(* IEC 61131-3 sources: elnaProjects/ElpcLogic/PomarKc7Unchanged/build_USO_ecl, 1 file *)

(* ---- plc.st ---- *)
TYPE
  TItemAIN : STRUCT
    wFlags : UINT := 0;
    wReserved : UINT := 0;
    dblValue : LREAL := 0.0;
    nanosec : ULINT := 0;
    reserve : ULINT := 0;
  END_STRUCT;
  TYPE_ReliableBit : STRUCT
    value : BOOL;
    reliability : BOOL;
    _inversed : BOOL;
  END_STRUCT;
  TItemDIN : STRUCT
    wFlags : UINT := 0;
    wValue : UINT := 0;
    nanosec : ULINT := 0;
    reserve : ULINT := 0;
  END_STRUCT;
  struct_DI : STRUCT
    imit : BOOL;
    value : WORD;
    reliability : WORD;
    bits : ARRAY [0..15] OF TYPE_ReliableBit;
    blConnect : BOOL;
  END_STRUCT;
  TYPE_StatusAi : STRUCT
    NOTDEFINED : BYTE := 0;
    LL : BYTE := 1;
    HL : BYTE := 2;
    NOTRELIABLE : BYTE := 3;
    normal : BYTE := 4;
    LW : BYTE := 5;
    HW : BYTE := 6;
    LA : BYTE := 7;
    HA : BYTE := 8;
  END_STRUCT;
  TWordData : STRUCT
    wFlags : UINT := 0;
    wValue : UINT := 0;
  END_STRUCT;
  TDoubleData : STRUCT
    wFlags : UINT := 0;
    dblValue : LREAL := 0.0;
  END_STRUCT;
  TYPE_statusDualInput : STRUCT
    STATUS_NOTDEFINED : BYTE := 0;
    STATUS_ON : BYTE := 1;
    STATUS_OFF : BYTE := 2;
    STATUS_TRANSITIONAL : BYTE := 3;
    STATUS_ERROR : BYTE := 4;
  END_STRUCT;
  TYPE_CommandAnalog : STRUCT
    cmd_SetUstavki : WORD := 1;
    cmd_SetRemont : WORD := 2;
    cmd_ResetRemont : WORD := 3;
    cmd_kvitNotReliable : WORD := 4;
  END_STRUCT;
  struct_AI : STRUCT
    value : LREAL;
    status : DWORD;
    interval : BYTE;
    inCommand : WORD;
    blConnect : BOOL;
    dLL : LREAL;
    dHL : LREAL;
    dLA : LREAL;
    dHA : LREAL;
    dLW : LREAL;
    dHW : LREAL;
    LL : LREAL;
    HL : LREAL;
    LA : LREAL;
    HA : LREAL;
    LW : LREAL;
    HW : LREAL;
    ISVALIDREF_LA : BOOL;
    ISVALIDREF_HA : BOOL;
    ISVALIDREF_LW : BOOL;
    ISVALIDREF_HW : BOOL;
    inpLL : LREAL;
    inpHL : LREAL;
    CurrentShotCircuit : LREAL;
    CurrentBreakCircuit : LREAL;
    maxChangeSpeed : LREAL;
    maxChangeSpeedDown : LREAL;
    ChangeSpeed : LREAL;
    histeresis : LREAL;
    aperturFilter : LREAL;
    exponentialFilter : LREAL;
    rassoglasovanie : LREAL;
    OpcCommandsDisabled : BOOL;
    Disabled_LA : BOOL;
    Disabled_HA : BOOL;
    Disabled_LW : BOOL;
    Disabled_HW : BOOL;
    delayLA : TIME;
    delayLW : TIME;
    delayHW : TIME;
    delayHA : TIME;
    minValue_ISVALIDREF : BOOL;
    maxValue_ISVALIDREF : BOOL;
    minValue : LREAL;
    maxValue : LREAL;
    inOpcCommandsDisabled : BOOL;
    imit : BOOL;
    remont : BOOL;
    NS : BOOL;
    NS_Min : BOOL;
    NS_Max : BOOL;
    inCommand_Alg : WORD;
    inCommand_ARM : WORD;
    dMaxChangeSpeed : LREAL;
    dMaxChangeSpeedDown : LREAL;
  END_STRUCT;
  AiConfig : STRUCT
    T_obmotki_fazy_1_k : struct_AI;
    T_aktivnogo_zheleza_statora_1_k : struct_AI;
    T_obmotki_fazy_2_k : struct_AI;
    T_aktivnogo_zheleza_statora_2_k : struct_AI;
    T_obmotki_fazy_3_k : struct_AI;
    T_aktivnogo_zheleza_statora_3_k : struct_AI;
    T_masla_v_maslobake : struct_AI;
    T_perednego_opornogo_podshipnika_dvigatelia_t1 : struct_AI;
    T_zadnego_opornogo_podshipnika_dvigatelia_t2 : struct_AI;
    T_masla_na_slive_perednego_opornogo_podshipnika_dvigatelia : struct_AI;
    T_masla_na_slive_zadnego_opornogo_podshipnika_dvigatelia : struct_AI;
    T_podshipnika_reduktora_t1 : struct_AI;
    T_podshipnika_reduktora_t2 : struct_AI;
    T_podshipnika_reduktora_t3 : struct_AI;
    T_podshipnika_reduktora_t4 : struct_AI;
    T_opornogo_podshipnika_nagnetatelia_t1 : struct_AI;
    T_opornogo_podshipnika_nagnetatelia_t2 : struct_AI;
    T_opornogo_podshipnika_nagnetatelia_t3 : struct_AI;
    T_oporno_upornogo_podshipnika_nagnetatelia_t4 : struct_AI;
    T_masla_do_AVOM : struct_AI;
    T_masla_posle_AVOM : struct_AI;
    T_gaz_in_nagnetatelia : struct_AI;
    T_gaz_out_nagnetatelia : struct_AI;
    T_hotAir_dvigatelia_t1 : struct_AI;
    T_clodAir_dvigatelia_t1 : struct_AI;
    dPmaslo_gaz : struct_AI;
    dP_gaza_na_konfuzore_nagnetatelia : struct_AI;
    P_masla_uplotneniia : struct_AI;
    P_gaza_na_vkhode_nagnetatelia : struct_AI;
    P_gaza_na_vykhode_nagnetatelia : struct_AI;
    P_masla_smazki_nizkoe : struct_AI;
    P_masla_smazki_srednee_posle_nasosov : struct_AI;
    Vibratciia_STD_t1 : struct_AI;
    Vibratciia_STD_t2 : struct_AI;
    Vibratciia_rotora_nagnetatelia_t1 : struct_AI;
    Vibratciia_rotora_nagnetatelia_t2 : struct_AI;
    Vibratciia_rotora_nagnetatelia_t3 : struct_AI;
    Vibratciia_rotora_nagnetatelia_t4 : struct_AI;
    Osevoi_sdvig_rotora_nagnetatelia : struct_AI;
    Uroven_masla_v_maslobake : struct_AI;
    Tok_vozbuzhdeniia_vozbuditelia : struct_AI;
    Tok_statora_elektrodvigatelia : struct_AI;
    Aktivnaia_moshchnost : struct_AI;
    Reaktivnaia_moshchnost : struct_AI;
    VoltageSHU_osnovnoi_vvod : struct_AI;
    VoltageSHU_rezervnyi_vvod : struct_AI;
    Rashod : struct_AI;
    Zapas : struct_AI;
    T_vnytri_shkafa : struct_AI;
  END_STRUCT;
  TYPE_AnalogLimitFlags : STRUCT
    NONE : BYTE := 0;
    LL : BYTE := 16#1;
    LW : BYTE := 16#2;
    HW : BYTE := 16#4;
    LA : BYTE := 16#8;
    HA : BYTE := 16#10;
    HL : BYTE := 16#20;
    SipUP : BYTE := 16#40;
    SipDown : BYTE := 16#80;
  END_STRUCT;
  DiConfig : STRUCT
    di_0 : struct_DI;
    di_1 : struct_DI;
    di_2 : struct_DI;
    di_3 : struct_DI;
    di_4 : struct_DI;
    di_5 : struct_DI;
    di_6 : struct_DI;
    di_7 : struct_DI;
    di_8 : struct_DI;
    di_9 : struct_DI;
    di_10 : struct_DI;
    di_11 : struct_DI;
    di_12 : struct_DI;
    di_13 : struct_DI;
    di_14 : struct_DI;
    di_15 : struct_DI;
  END_STRUCT;
  TYPE_commandDualInput : STRUCT
    CMD_ON : BYTE := 1;
    CMD_OFF : BYTE := 2;
    CMD_RESET : BYTE := 3;
  END_STRUCT;
  struct_DO : STRUCT
    imit : BOOL;
    blConnect : BOOL;
    value : WORD;
    bits : ARRAY [0..15] OF BOOL;
  END_STRUCT;
  DOconfig : STRUCT
    do_0 : struct_DO;
    do_1 : struct_DO;
    do_2 : struct_DO;
    do_3 : struct_DO;
    do_4 : struct_DO;
    do_5 : struct_DO;
    do_6 : struct_DO;
    do_7 : struct_DO;
    gpio_out : struct_DO;
  END_STRUCT;
  struct_AO : STRUCT
    nValue : LREAL;
    blConnect : BOOL;
    outLL : LREAL;
    outHL : LREAL;
    newLL : LREAL;
    newHL : LREAL;
    newLL_ISVALIDREF : BOOL;
    newHL_ISVALIDREF : BOOL;
    inCommand : WORD;
    Value : LREAL;
    status : DWORD;
    LL : LREAL;
    HL : LREAL;
    OpcCommandsDisabled : BOOL;
  END_STRUCT;
  AOConfig : STRUCT
    Reserv_AO_1 : struct_AO;
    Reserv_AO_2 : struct_AO;
  END_STRUCT;
  struct_singleSignal : STRUCT
    reliability : BOOL;
    inverse : BOOL;
    DelayOn : TIME;
    DelayOff : TIME;
    Q : BOOL;
    status : DWORD;
    Disabled_Sig : BOOL;
  END_STRUCT;
  IM_singleSignals : STRUCT
    dP_gazgaz_Kran1 : struct_singleSignal;
    OsevoiSdvig_pravo : struct_singleSignal;
    OsevoiSdvig_levo : struct_singleSignal;
    dP_oilgaz_low : struct_singleSignal;
    P_oil_low : struct_singleSignal;
    KZ_10kv : struct_singleSignal;
    Vozb_ProboiVentila : struct_singleSignal;
    Vozb_AsinchHod : struct_singleSignal;
    Vozb_ReSynchronize : struct_singleSignal;
    Vozb_ControlVozbuditela : struct_singleSignal;
    NS_ForsingVozbugdenia : struct_singleSignal;
    NS_Vozbyditela : struct_singleSignal;
    Vozb_AVR_off : struct_singleSignal;
    Vozb_AutoUprVozbuditela_off : struct_singleSignal;
    Vozb_KontaktorON : struct_singleSignal;
    Vozb_Overload : struct_singleSignal;
    AO_KC : struct_singleSignal;
    AOGPA_PRU : struct_singleSignal;
    BEO_Ready : struct_singleSignal;
    BEO_Srabat : struct_singleSignal;
    BEO_ON_knopkaSHU : struct_singleSignal;
    BEO_ON_knopkaPRU : struct_singleSignal;
    NOGPA_knopkaSHU : struct_singleSignal;
    AOGPA_knopkaSHU : struct_singleSignal;
    DverShkafaOtkryta : struct_singleSignal;
    QF1_on : struct_singleSignal;
    QF2_on : struct_singleSignal;
    QF23_on : struct_singleSignal;
    QF4_QF5_on : struct_singleSignal;
    QF6_QF7_on : struct_singleSignal;
    QF8_QF9_on : struct_singleSignal;
    QF10_QF11_on : struct_singleSignal;
    QF12_QF13_on : struct_singleSignal;
    QF14_QF15_on : struct_singleSignal;
    QF22_on : struct_singleSignal;
    NS_G1_G2 : struct_singleSignal;
    NS_G3_G4 : struct_singleSignal;
    NS_G15_G16 : struct_singleSignal;
    NS_G17 : struct_singleSignal;
    NS_G5_G6 : struct_singleSignal;
    NS_G7_G8 : struct_singleSignal;
    NS_G18_G19 : struct_singleSignal;
    NS_G10_G11 : struct_singleSignal;
    NS_G13_G14 : struct_singleSignal;
  END_STRUCT;
  struct_singleOutput : STRUCT
    wait_time : TIME;
    inCommand : WORD;
    inOpcCommandsDisabled : BOOL;
    Q : BOOL;
    status : DWORD;
    OpcCommandsDisabled : BOOL;
    inCommand_Alg : WORD;
    inCommand_ARM : WORD;
  END_STRUCT;
  IM_singleOutputs : STRUCT
    Lampa_NO : struct_singleOutput;
    VzvodBREO : struct_singleOutput;
    AO_GPA : struct_singleOutput;
    SbrosBREO : struct_singleOutput;
    IndikicijaPS_fonar : struct_singleOutput;
    IndikicijaAS_fonar : struct_singleOutput;
    mv_off_KNA : struct_singleOutput;
  END_STRUCT;
  struct_Kran : STRUCT
    inCommand : WORD;
    status : DWORD;
    onStatus : BYTE;
    inOpcCommandsDisabled : BOOL;
    sdvig : BOOL;
    Ns : BOOL;
    Dp : BOOL;
    CommandFault : BOOL;
    Accident : BOOL;
    Auto : BOOL;
    Manual : BOOL;
    Local : BOOL;
    Distance : BOOL;
    ErrorPowerOff : BOOL;
    ErrorBlock : BOOL;
    So : BOOL;
    Sz : BOOL;
    OpcCommandsDisabled : BOOL;
    lastCmdIsOn : BOOL;
    ISVALIDREF_statOn : BOOL;
    ISVALIDREF_statOff : BOOL;
    ISVALIDREF_cmdOn : BOOL;
    ISVALIDREF_cmdOff : BOOL;
    ISVALIDREF_inSo : BOOL;
    ISVALIDREF_inSz : BOOL;
    ISVALIDREF_inDp : BOOL;
    continueHoldCommand : TIME;
    inCommand_Alg : WORD;
    inCommand_ARM : WORD;
    cmdOn : BOOL;
    cmdOff : BOOL;
    reliability : BOOL;
  END_STRUCT;
  struct_OilPump : STRUCT
    inCommand : WORD;
    inCommand_Alg : WORD;
    inCommand_ARM : WORD;
    status : DWORD;
    onStatus : BYTE;
    inOpcCommandsDisabled : BOOL;
    sdvig : BOOL;
    Ns : BOOL;
    CommandFault : BOOL;
    Accident : BOOL;
    Local : BOOL;
    Distance : BOOL;
    BreakCmdOn : BOOL;
    BreakCmdOff : BOOL;
    OpcCommandsDisabled : BOOL;
    lastCmdIsOn : BOOL;
    ISVALIDREF_statOn : BOOL;
    ISVALIDREF_statOff : BOOL;
    ISVALIDREF_cmdOn : BOOL;
    ISVALIDREF_cmdOff : BOOL;
    ISVALIDREF_inBreakCmdOn : BOOL;
    ISVALIDREF_inBreakCmdOff : BOOL;
    inBlocked : BOOL;
    Blocked : BOOL;
    Osnovnoy : BOOL;
    Rezervny : BOOL;
    cmdOn : BOOL;
    cmdOff : BOOL;
    reliability : BOOL;
  END_STRUCT;
  struct_Switch : STRUCT
    inCommand : WORD;
    status : DWORD;
    onStatus : BYTE;
    inOpcCommandsDisabled : BOOL;
    sdvig : BOOL;
    Ns : BOOL;
    CommandFault : BOOL;
    Accident : BOOL;
    Auto : BOOL;
    Manual : BOOL;
    Local : BOOL;
    Distance : BOOL;
    ErrorPowerOff : BOOL;
    ErrorBlock : BOOL;
    BreakCmdOn : BOOL;
    BreakCmdOff : BOOL;
    OpcCommandsDisabled : BOOL;
    lastCmdIsOn : BOOL;
    ISVALIDREF_statOn : BOOL;
    ISVALIDREF_statOff : BOOL;
    ISVALIDREF_cmdOn : BOOL;
    ISVALIDREF_cmdOff : BOOL;
    ISVALIDREF_inBreakCmdOn : BOOL;
    ISVALIDREF_inBreakCmdOff : BOOL;
    inCommand_Alg : WORD;
    inCommand_ARM : WORD;
    cmdOn : BOOL;
    cmdOff : BOOL;
    reliability : BOOL;
  END_STRUCT;
  struct_SectionSwitch : STRUCT
    inCommand : WORD;
    status : DWORD;
    onStatus : BYTE;
    inOpcCommandsDisabled : BOOL;
    sdvig : BOOL;
    Ns : BOOL;
    CommandFault : BOOL;
    Accident : BOOL;
    Local : BOOL;
    Distance : BOOL;
    OpcCommandsDisabled : BOOL;
    lastCmdIsOn : BOOL;
    offKNA : BOOL;
    basketStatus : BYTE;
    ISVALIDREF_statOn : BOOL;
    ISVALIDREF_statOff : BOOL;
    ISVALIDREF_cmdOn : BOOL;
    ISVALIDREF_cmdOff : BOOL;
    ISVALIDREF_inBreakCmdOn : BOOL;
    ISVALIDREF_inBreakCmdOff : BOOL;
    BreakCmdOn : BOOL;
    BreakCmdOff : BOOL;
    ISVALIDREF_basketRolledIn : BOOL;
    ISVALIDREF_basketRolledOut : BOOL;
    ISVALIDREF_basketTest : BOOL;
    inCommand_Alg : WORD;
    inCommand_ARM : WORD;
    cmdOn : BOOL;
    cmdOff : BOOL;
    reliability : BOOL;
  END_STRUCT;
  struct_ReserveIM : STRUCT
    var1 : BOOL;
    var2 : BOOL;
  END_STRUCT;
  struct_ReserveIM2 : STRUCT
    var1 : BOOL;
    var2 : BOOL;
  END_STRUCT;
  struct_AnalogParametr : STRUCT
    inCommand : WORD;
    inCommand_Alg : WORD;
    inCommand_ARM : WORD;
    status : DWORD;
    newValue : LREAL;
    currentValue : LREAL;
    minVal : LREAL;
    maxVal : LREAL;
    maxStep : LREAL;
    minVal_ISVALIDREF : BOOL;
    maxVal_ISVALIDREF : BOOL;
    maxStep_ISVALIDREF : BOOL;
    inOpcCommandsDisabled : BOOL;
    Value : LREAL;
    isValidValue : BOOL;
    OpcCommandsDisabled : BOOL;
  END_STRUCT;
  struct_DiscretParametr : STRUCT
    newValue : UINT;
    currentValue : UINT;
    inOpcCommandsDisabled : BOOL;
    inCommand : WORD;
    inCommand_Alg : WORD;
    inCommand_ARM : WORD;
    status : DWORD;
    OpcCommandsDisabled : BOOL;
    Value : UINT;
  END_STRUCT;
  ImConfig : STRUCT
    Kran1 : struct_Kran;
    Kran2 : struct_Kran;
    Kran3b : struct_Kran;
    Kran4 : struct_Kran;
    Kran5 : struct_Kran;
    Kran6 : struct_Kran;
    nu1 : struct_OilPump;
    nu2 : struct_OilPump;
    pns : struct_Switch;
    v1_Avom : struct_Switch;
    v2_Avom : struct_Switch;
    mv : struct_SectionSwitch;
    Ten : struct_Switch;
    Reserve_IM1 : struct_ReserveIM;
    Reserve_IM2 : struct_ReserveIM2;
    SingleSignals : IM_singleSignals;
    SingleOutputs : IM_singleOutputs;
    AutoAvom_onTemp1 : struct_AnalogParametr;
    AutoAvom_onTemp2 : struct_AnalogParametr;
    AutoAvom_hysteresis : struct_AnalogParametr;
    TypeSwitch : struct_DiscretParametr;
    AutoPns_UstRun : struct_AnalogParametr;
    AutoPns_UstStop : struct_AnalogParametr;
    AutoNU_mainNU : struct_DiscretParametr;
    PuskOilSystem_UstdPmg : struct_AnalogParametr;
    AutoTen_offTemperature : struct_AnalogParametr;
    AutoNU_Ust_Swap : struct_AnalogParametr;
    testdPmg_Ust_dPLow : struct_AnalogParametr;
    AntiPompag_UgolVNA : struct_AnalogParametr;
    AntiPompag_K : struct_AnalogParametr;
    AntiPompag_A : struct_AnalogParametr;
    AntiPompag_y0 : struct_AnalogParametr;
  END_STRUCT;
  struct_DualStateIm : STRUCT
    inCommand : WORD;
    status : DWORD;
    onStatus : BYTE;
    inOpcCommandsDisabled : BOOL;
    sdvig : BOOL;
    Ns : BOOL;
    CommandFault : BOOL;
    Accident : BOOL;
    OpcCommandsDisabled : BOOL;
    lastCmdIsOn : BOOL;
    ISVALIDREF_statOn : BOOL;
    ISVALIDREF_statOff : BOOL;
    ISVALIDREF_cmdOn : BOOL;
    ISVALIDREF_cmdOff : BOOL;
    inCommand_Alg : WORD;
    inCommand_ARM : WORD;
    cmdOn : BOOL;
    cmdOff : BOOL;
    reliability : BOOL;
  END_STRUCT;
  TYPE_ProtectionTags : STRUCT
    NOTHING : BYTE := 0;
    AOB : BYTE := 1;
    AOS : BYTE := 2;
    AOPOJ : BYTE := 3;
  END_STRUCT;
  TYPE_basketStats : STRUCT
    BASKET_NOTDEFINED : BYTE := 0;
    BASKET_ROLLEDIN : BYTE := 1;
    BASKET_ROLLEDOUT : BYTE := 2;
    BASKET_TRANSITIONAL : BYTE := 3;
    BASKET_ERROR : BYTE := 4;
    BASKET_TEST : BYTE := 5;
  END_STRUCT;
  struct_AiProtection : STRUCT
    controlLimit : BYTE;
    delay : TIME;
    inTag : BYTE;
    inRunOnStart : BOOL;
    inCanRun : BOOL;
    inOpcCommandsDisabled : BOOL;
    inCommand : WORD;
    inCommand_Alg : WORD;
    inCommand_ARM : WORD;
    Tag : BYTE;
    status : DWORD;
    CanRun : BOOL;
    OpcCommandsDisabled : BOOL;
    isRunning : BOOL;
    HasError : BOOL;
    isEnded : BOOL;
    Remont : BOOL;
    Check : BOOL;
    Signaling : BOOL;
    SignalingTP : BOOL;
    RunOnStart : BOOL;
  END_STRUCT;
  struct_DiProtection : STRUCT
    delay : TIME;
    inTag : BYTE;
    inRunOnStart : BOOL;
    inCanRun : BOOL;
    inOpcCommandsDisabled : BOOL;
    inCommand : WORD;
    inCommand_Alg : WORD;
    inCommand_ARM : WORD;
    Tag : BYTE;
    status : DWORD;
    CanRun : BOOL;
    OpcCommandsDisabled : BOOL;
    isRunning : BOOL;
    HasError : BOOL;
    isEnded : BOOL;
    Remont : BOOL;
    Check : BOOL;
    Signaling : BOOL;
    SignalingTP : BOOL;
    RunOnStart : BOOL;
  END_STRUCT;
  ProtectionsConfig : STRUCT
    T_perednego_opornogo_podshipnika_dvigatelia_t1_HA : struct_AiProtection;
    T_zadnego_opornogo_podshipnika_dvigatelia_t2_HA : struct_AiProtection;
    T_podshipnika_reduktora_t1_HA : struct_AiProtection;
    T_podshipnika_reduktora_t2_HA : struct_AiProtection;
    T_podshipnika_reduktora_t3_HA : struct_AiProtection;
    T_podshipnika_reduktora_t4_HA : struct_AiProtection;
    T_opornogo_podshipnika_nagnetatelia_t1_HA : struct_AiProtection;
    T_opornogo_podshipnika_nagnetatelia_t2_HA : struct_AiProtection;
    T_opornogo_podshipnika_nagnetatelia_t3_HA : struct_AiProtection;
    T_opornoupornogo_podshipnika_nagnetatelia_t4_HA : struct_AiProtection;
    T_gaza_na_vykhode_nagnetatelia_HA : struct_AiProtection;
    dP_maslogaz_LA : struct_AiProtection;
    P_masla_smazki_nizkoe_LA : struct_AiProtection;
    Vibratciia_STD_t1_HA : struct_AiProtection;
    Vibratciia_STD_t2_HA : struct_AiProtection;
    Vibratciia_rotora_nagnetatelia_t1_HA : struct_AiProtection;
    Vibratciia_rotora_nagnetatelia_t2_HA : struct_AiProtection;
    Vibratciia_rotora_nagnetatelia_t3_HA : struct_AiProtection;
    Vibratciia_rotora_nagnetatelia_t4_HA : struct_AiProtection;
    Osevoi_sdvig_rotora_nagnetatelia_HA : struct_AiProtection;
    Uroven_masla_v_maslobake_LA : struct_AiProtection;
    OsevojSdvigPravyjDi : struct_DiProtection;
    OsevojSdvigLevyjDi : struct_DiProtection;
    dP_masloGaz_LowDI : struct_DiProtection;
    DavlenieMaslaSmazkiDi : struct_DiProtection;
    mvOff : struct_DiProtection;
    NeispravnostVozbuzhdenijaDi : struct_DiProtection;
    AO_KC : struct_DiProtection;
    AO_PRU : struct_DiProtection;
    AO_SHU : struct_DiProtection;
    Srab_BEAO : struct_DiProtection;
    EAO_PRU : struct_DiProtection;
    BEAO_knSHU : struct_DiProtection;
    Kran1sdvig : struct_DiProtection;
    Kran2sdvig : struct_DiProtection;
  END_STRUCT;
  TYPE_ModeGpa : STRUCT
    MODE_NOTDEFINED : UINT := 0;
    MODE_REMONT : UINT := 1;
    MODE_STOP : UINT := 2;
    MODE_READY : UINT := 3;
    MODE_PUSKV : UINT := 4;
    MODE_PUSKK : UINT := 5;
    MODE_TESTDPMG : UINT := 6;
    MODE_TESTPMS : UINT := 7;
    MODE_APUSK : UINT := 8;
    MODE_MPUSK : UINT := 9;
    MODE_WORK_Ring : UINT := 10;
    MODE_WORK_Line : UINT := 11;
    MODE_NO : UINT := 12;
    MODE_AO : UINT := 13;
    MODE_EO : UINT := 14;
    MODE_TESTIM : UINT := 15;
    MODE_TESTAZ : UINT := 16;
  END_STRUCT;
  TYPE_DualStateImAction : (_on, _off) := _on;
  TYPE_PhaseAlgoritmAction : (_run, _reset) := _run;
  TYPE_Answers : STRUCT
    ANS_NONE : UINT := 0;
    ANS_YES : UINT := 1;
    ANS_NO : UINT := 2;
    ANS_CANCEL : UINT := 4;
    ANS_RETRY : UINT := 8;
  END_STRUCT;
  struct_Alg : STRUCT
    inRunOnStart : BOOL;
    inCanRun : BOOL;
    inHasError : BOOL;
    inEnded : BOOL;
    inOpcCommandsDisabled : BOOL;
    inCommand : WORD;
    inCommand_ARM : WORD;
    inCommand_Alg : WORD;
    status : DWORD;
    CanRun : BOOL;
    OpcCommandsDisabled : BOOL;
    isRuning : BOOL;
    HasError : BOOL;
    isEnded : BOOL;
    RunOnStart : BOOL;
    Start : DWORD;
    Error : DWORD;
    Top : DWORD;
  END_STRUCT;
  AlgoritmsConfig : STRUCT
    autoNu : struct_Alg;
    AutoPns : struct_Alg;
    AutoAvom : struct_Alg;
    AutoTen : struct_Alg;
    AntiPompag : struct_Alg;
    testIm : struct_Alg;
    TestProtection : struct_Alg;
    Remont : struct_Alg;
    ppu : struct_Alg;
    puskOilSystem : struct_Alg;
    engineRun : struct_Alg;
    filling : struct_Alg;
    LineToRing : struct_Alg;
    RingToLine : struct_Alg;
    Apusk : struct_Alg;
    SemiAutoPusk : struct_Alg;
    no : struct_Alg;
    vibegPNS : struct_Alg;
    ao : struct_Alg;
    testPms : struct_Alg;
    testdPmg : struct_Alg;
    puskV : struct_Alg;
    puskK : struct_Alg;
  END_STRUCT;
  TYPE_CommandsPotectionsManager : STRUCT
    RestartAllSignaling : BYTE := 1;
    RestartAllProtections : BYTE := 2;
    CheckProtections : BYTE := 3;
    ResetAllProtections : BYTE := 4;
  END_STRUCT;
  struct_ProtectionsManager : STRUCT
    inCommand : BYTE;
    protectionInRemont : BOOL;
  END_STRUCT;
  struct_AlgoritmsManager : STRUCT
    mode : UINT;
    narabotka : UINT;
    nMode : UINT;
    AnalogsPs : BOOL;
    DiscretPS : BOOL;
    ProtectionSignaling : BOOL;
  END_STRUCT;
  struct_AlgTimers : STRUCT
    AutoPns_OffTimer : UINT;
    AutoPns_OnTimer : UINT;
    vibegPNS_Timer : UINT;
    NO_waitCloseKran : UINT;
    AO_waitKran : UINT;
    testPms_BreakTest : UINT;
    testdPmg_BreakTest : UINT;
    puskOilSystem_BreakPuskTimer_Poil : UINT;
    engineRun_BreakPuskTimer : UINT;
    filling_BreakPuskTimer : UINT;
    filling_waitAfterKran4 : UINT;
    filling_waitAfterKran5 : UINT;
    puskK_wait720 : UINT;
    puskV_wait600 : UINT;
  END_STRUCT;
  struct_PhaseAlgoritm : STRUCT
    run : BOOL;
    reset : BOOL;
    start : BOOL;
    error : BOOL;
    top : BOOL;
    startStatus : DWORD;
    errorStatus : DWORD;
    topStatus : DWORD;
  END_STRUCT;
  struct_Question : STRUCT
    AnswerVariants : UINT;
    inCommand : WORD;
    ask : BOOL;
    reset : BOOL;
    status : DWORD;
    answer : UINT;
    OpcCommandsDisabled : BOOL;
    inOpcCommandsDisabled : BOOL;
  END_STRUCT;
  AlgoritmsQuestions : STRUCT
    vibegPNS_algContinue : struct_Question;
    testPms_algContinue : struct_Question;
    testdPmg_algContinue : struct_Question;
    puskK_questionFilling : struct_Question;
    puskK_questionUnload : struct_Question;
    puskV_questionEngine : struct_Question;
    puskV_questionMVoff : struct_Question;
    SemiAutoPusk_cmdRun1ph : struct_Question;
    SemiAutoPusk_cmdRun2ph : struct_Question;
    SemiAutoPusk_cmdRun3ph : struct_Question;
    SemiAutoPusk_cmdRun4ph : struct_Question;
  END_STRUCT;
  TYPE_TableRec : STRUCT
    x : REAL;
    y : REAL;
  END_STRUCT;
END_TYPE

FUNCTION_BLOCK fb_Timings
  VAR_EXTERNAL CONSTANT
    req_Cycle : REAL;
  END_VAR
  VAR_EXTERNAL
    gF_T_100mSec : BOOL;
    gT_1Sec : BOOL;
    gF_T_1Sec : BOOL;
    gT_1Min : BOOL;
    gR_T_1Min : BOOL;
    gF_T_1Min : BOOL;
    del_T : REAL;
    cur_Cycle : REAL;
  END_VAR
  VAR
    Tmr_100_ms : REAL;
  END_VAR
  VAR_EXTERNAL
    T_1SEC : REAL;
  END_VAR
  VAR
    Tmr_1_s : REAL;
    Tmr_1_min : REAL;
  END_VAR

  (* Обработка времени. *)
  Tmr_100_ms := Tmr_100_ms + cur_Cycle;
  gF_T_100mSec := FALSE;
  IF Tmr_100_ms >= 0.1 THEN Tmr_100_ms := 0.0; gF_T_100mSec := TRUE; END_IF;

  Tmr_1_s := Tmr_1_s + cur_Cycle;
  gF_T_1Sec := FALSE;
  IF Tmr_1_s >= 1.0 THEN Tmr_1_s := 0.0; gF_T_1Sec := TRUE; END_IF;

  T_1SEC := T_1SEC + cur_Cycle;
  gT_1Sec := FALSE;
  IF T_1SEC >= 2.0 THEN T_1SEC := 0.0;
    ELSIF T_1SEC >= 1.0 THEN gT_1Sec := TRUE; END_IF;

  IF Tmr_1_min > 60.0 THEN
      Tmr_1_min := 0.0; gF_T_1Min := gT_1Min; gT_1Min := NOT gT_1Min; gR_T_1Min := gT_1Min;
    ELSE
      Tmr_1_min := Tmr_1_min + cur_Cycle; gR_T_1Min := FALSE; gF_T_1Min := FALSE;
  END_IF;
  del_T:= cur_Cycle;
END_FUNCTION_BLOCK

FUNCTION_BLOCK fb_AI_Init
  VAR_INPUT
    data_Ini : BOOL;
    dLL : LREAL;
    dHL : LREAL;
    dLA : LREAL;
    dHA : LREAL;
    dLW : LREAL;
    dHW : LREAL;
    ISVALIDREF_LA : BOOL := False;
    ISVALIDREF_HA : BOOL := False;
    ISVALIDREF_LW : BOOL := False;
    ISVALIDREF_HW : BOOL := False;
    delayLA : TIME := T#0S;
    delayLW : TIME := T#0S;
    delayHW : TIME := T#0S;
    delayHA : TIME := T#0S;
    inpLL : LREAL := 4000.0;
    inpHL : LREAL := 20000.0;
    CurrentShotCircuit : LREAL := 21000.0;
    CurrentBreakCircuit : LREAL := 3700.0;
    dMaxChangeSpeed : LREAL;
    dMaxChangeSpeedDown : LREAL;
    histeresis : LREAL;
    aperturFilter : LREAL;
    exponentialFilter : LREAL;
    rassoglasovanie : LREAL;
    inOpcCommandsDisabled : BOOL;
  END_VAR
  VAR_IN_OUT
    strAI : struct_AI;
  END_VAR
  VAR_OUTPUT
    Init : BOOL := FALSE;
  END_VAR

  (*****            Функциональный блок переинициализации структуры-дескриптора канала аналогового ввода.            *****)
       Init := false;

      IF data_Ini THEN                            (* Параметрам требуется переинициализация. *)
          strAI.dLL                := dLL;
          strAI.dHL                := dHL;
          strAI.dLA                := dLA;
          strAI.dHA                := dHA;
          strAI.dLW                := dLW;
          strAI.dHW                := dHW;
          strAI.ISVALIDREF_LA      := ISVALIDREF_LA;
          strAI.ISVALIDREF_HA      := ISVALIDREF_HA;
          strAI.ISVALIDREF_LW      := ISVALIDREF_LW;
          strAI.ISVALIDREF_HW      := ISVALIDREF_HW;
          strAI.delayLA            := delayLA;
          strAI.delayLW            := delayLW;
          strAI.delayHW            := delayHW;
          strAI.delayHA            := delayHA;
          strAI.inpLL              := inpLL;
          strAI.inpHL              := inpHL;
          strAI.CurrentShotCircuit := CurrentShotCircuit;
          strAI.CurrentBreakCircuit:= CurrentBreakCircuit;
          strAI.dMaxChangeSpeed     := dMaxChangeSpeed;
          strAI.dMaxChangeSpeedDown := dMaxChangeSpeedDown;
          strAI.histeresis         := histeresis;
          strAI.aperturFilter      := aperturFilter;
          strAI.exponentialFilter  := exponentialFilter;
          strAI.rassoglasovanie    := rassoglasovanie;
          strAI.rassoglasovanie    := rassoglasovanie;

          data_Ini:=false;
          Init := TRUE;
       END_IF;
    IF Init THEN
          dLL:= 0.0;
          dHL:= 0.0;
          dLA:= 0.0;
          dHA:= 0.0;
          dLW:= 0.0;
          dHW:= 0.0;
          inpLL:= 4000.0;
          inpHL:= 20000.0;
          CurrentShotCircuit:= 21000.0;
          CurrentBreakCircuit:= 3700.0;
          ISVALIDREF_LA:= false;
          ISVALIDREF_HA:= false;
          ISVALIDREF_LW:= false;
          ISVALIDREF_HW:= false;
          delayLA:= T#0S;
          delayLW:= T#0S;
          delayHW:= T#0S;
          delayHA:= T#0S;
          dMaxChangeSpeed:= 0.0;
          dMaxChangeSpeedDown:= 0.0;
          histeresis:= 0.0;
          aperturFilter:= 0.0;
          exponentialFilter:= 0.0;
          rassoglasovanie:= 0.0;
        END_IF;
END_FUNCTION_BLOCK

FUNCTION_BLOCK proc_AI_Init
  VAR_INPUT
    init : BOOL;
  END_VAR
  VAR
    stAI_Ini : fb_AI_Init;
    inits : UINT;
  END_VAR
  VAR_INPUT
    initiales : UINT;
  END_VAR
  VAR_EXTERNAL
    ai : AiConfig;
  END_VAR

  (* Инициализация начало. Входные аналоговые параметры *)

  inits := 0; (* Флаг необходимости инициализации структур-дескрипторов *)

  (********************************************* Модуль A1-4 ******************************************************)
  (* [A1-4, AI0-0] Т обмотки фазы 1 канал *)
  stAI_Ini(data_Ini := TRUE, dLL := 0.0, dHL := 180.0,
  strAI := ai.T_obmotki_fazy_1_k);
  inits := inits + BOOL_TO_UINT(stAI_Ini.Init);

  (* [A1-4, AI0-1] Т активного железа статора 1 канал *)
  stAI_Ini(data_Ini := TRUE,  dLL := 0.0, dHL := 180.0, strAI := ai.T_aktivnogo_zheleza_statora_1_k);
  inits := inits + BOOL_TO_UINT(stAI_Ini.Init);

  (* [A1-4, AI0-2] ТТ обмотки фазы 2 канал *)
  stAI_Ini(data_Ini := TRUE,  dLL := 0.0, dHL :=180.0, strAI := ai.T_obmotki_fazy_2_k);
  inits := inits + BOOL_TO_UINT(stAI_Ini.Init);

  (* [A1-4, AI0-3] Т активного железа статора 2 канал *)
  stAI_Ini(data_Ini := TRUE,  dLL := 0.0, dHL := 180.0, strAI := ai.T_aktivnogo_zheleza_statora_2_k);
  inits := inits + BOOL_TO_UINT(stAI_Ini.Init);

  (* [A1-4, AI0-4] Т обмотки фазы 3 канал *)
  stAI_Ini(data_Ini :=TRUE,  dLL := 0.0, dHL := 180.0, strAI := ai.T_obmotki_fazy_3_k);
  inits := inits + BOOL_TO_UINT(stAI_Ini.Init);

  (* [A1-4, AI0-5] Т активного железа статора 3 канал *)
  stAI_Ini(data_Ini := TRUE,  dLL := 0.0, dHL := 180.0, strAI := ai.T_aktivnogo_zheleza_statora_3_k);
  inits := inits + BOOL_TO_UINT(stAI_Ini.Init);

  (* [A1-4, AI0-6] Т масла в маслобаке } *)
  stAI_Ini(data_Ini := TRUE,  dLL := -50.0, dHL := 150.0,
  ISVALIDREF_LW := TRUE, ISVALIDREF_HW := TRUE, dLW := 20.0, dHW := 55.0,
  strAI := ai.T_masla_v_maslobake);
  inits := inits + BOOL_TO_UINT(stAI_Ini.Init);

  (********************************************** Модуль A1-5 *********************************************************)
  (* [A1-5, AI1-0]  Т переднего опорного подшипника двигателя, т.1 *)
  stAI_Ini(data_Ini := TRUE,  dLL := -50.0, dHL := 120.0,
  ISVALIDREF_HA := TRUE, ISVALIDREF_HW := TRUE, dHA := 85.0, dHW := 80.0,
  strAI := ai.T_perednego_opornogo_podshipnika_dvigatelia_t1);
  inits := inits + BOOL_TO_UINT(stAI_Ini.Init);

  (* [A1-5, AI1-1]  Т заднего опорного подшипника двигателя, т.2 *)
  stAI_Ini(data_Ini := TRUE,  dLL := -50.0, dHL := 120.0,
  ISVALIDREF_HA := TRUE, ISVALIDREF_HW := TRUE, dHA := 85.0, dHW := 80.0,
  strAI := ai.T_zadnego_opornogo_podshipnika_dvigatelia_t2);
  inits := inits + BOOL_TO_UINT(stAI_Ini.Init);

  (* [A1-5, AI1-2] Т масла на сливе переднего опорного подшипника двигателя *)
  stAI_Ini(data_Ini := TRUE,  dLL := -50.0, dHL := 150.0, strAI := ai.T_masla_na_slive_perednego_opornogo_podshipnika_dvigatelia);
  inits := inits + BOOL_TO_UINT(stAI_Ini.Init);

  (* [A1-5, AI1-3] Т масла на сливе заднего опорного подшипника двигателя *)
  stAI_Ini(data_Ini := TRUE,  dLL := -50.0, dHL := 150.0, strAI := ai.T_masla_na_slive_zadnego_opornogo_podshipnika_dvigatelia);
  inits := inits + BOOL_TO_UINT(stAI_Ini.Init);

  (* [A1-5, AI1-4]  Т подшипника редуктора, т1 *)
  stAI_Ini(data_Ini := TRUE,  dLL := -50.0, dHL := 150.0,
  ISVALIDREF_HA := TRUE, ISVALIDREF_HW := TRUE, dHA := 85.0, dHW := 80.0,
  strAI := ai.T_podshipnika_reduktora_t1);
  inits := inits + BOOL_TO_UINT(stAI_Ini.Init);

  (* [A1-5, AI1-5]  Т подшипника редуктора, т2 *)
  stAI_Ini(data_Ini := TRUE,  dLL := -50.0, dHL := 150.0,
  ISVALIDREF_HA := TRUE, ISVALIDREF_HW := TRUE, dHA := 85.0, dHW := 80.0,
  strAI := ai.T_podshipnika_reduktora_t2);
  inits := inits + BOOL_TO_UINT(stAI_Ini.Init);

  (* [A1-5, AI1-6]  Т подшипника редуктора, т3 *)
  stAI_Ini(data_Ini := TRUE,  dLL := -50.0, dHL := 150.0,
  ISVALIDREF_HA := TRUE, ISVALIDREF_HW := TRUE, dHA := 85.0, dHW := 80.0,
  strAI := ai.T_podshipnika_reduktora_t3);
  inits := inits + BOOL_TO_UINT(stAI_Ini.Init);

  (* [A1-5, AI1-7]  Т подшипника редуктора, т4 *)
  stAI_Ini(data_Ini := TRUE,  dLL := -50.0, dHL := 150.0,
  ISVALIDREF_HA := TRUE, ISVALIDREF_HW := TRUE, dHA := 85.0, dHW := 80.0,
  strAI := ai.T_podshipnika_reduktora_t4);
  inits := inits + BOOL_TO_UINT(stAI_Ini.Init);

  (********************************************** Модуль A1-6 *********************************************************)
  (* [A1-6, AI2-0]  Т опорного подшипника нагнетателя, т1 *)
  stAI_Ini(data_Ini := TRUE,  dLL := -50.0, dHL := 150.0,
  ISVALIDREF_HA := TRUE, ISVALIDREF_HW := TRUE, dHA := 85.0, dHW := 80.0,
  strAI := ai.T_opornogo_podshipnika_nagnetatelia_t1);
  inits := inits + BOOL_TO_UINT(stAI_Ini.Init);

  (* [A1-6, AI2-1]  Т опорного подшипника нагнетателя, т2 *)
  stAI_Ini(data_Ini := TRUE,  dLL := -50.0, dHL := 150.0,
  ISVALIDREF_HA := TRUE, ISVALIDREF_HW := TRUE, dHA := 85.0, dHW := 80.0,
  strAI := ai.T_opornogo_podshipnika_nagnetatelia_t2);
  inits := inits + BOOL_TO_UINT(stAI_Ini.Init);

  (* [A1-6, AI2-2]  Т опорного подшипника нагнетателя, т3 *)
  stAI_Ini(data_Ini := TRUE,  dLL := -50.0, dHL := 150.0,
  ISVALIDREF_HA := TRUE, ISVALIDREF_HW := TRUE, dHA := 85.0, dHW := 80.0,
  strAI := ai.T_opornogo_podshipnika_nagnetatelia_t3);
  inits := inits + BOOL_TO_UINT(stAI_Ini.Init);

  (* [A1-6, AI2-3]  Т опорно-упорного подшипника нагнетателя, т4 *)
  stAI_Ini(data_Ini := TRUE,  dLL := -50.0, dHL := 150.0,
  ISVALIDREF_HA := TRUE, ISVALIDREF_HW := TRUE, dHA := 85.0, dHW := 80.0,
  strAI := ai.T_oporno_upornogo_podshipnika_nagnetatelia_t4);
  inits := inits + BOOL_TO_UINT(stAI_Ini.Init);

  (* [A1-6, AI2-4] Т масла до АВОМ *)
  stAI_Ini(data_Ini := TRUE,  dLL := -50.0, dHL := 150.0, strAI := ai.T_masla_do_AVOM);
  inits := inits + BOOL_TO_UINT(stAI_Ini.Init);

  (* [A1-6, AI2-5] Т масла после АВОМ *)
  stAI_Ini(data_Ini := TRUE,  dLL := -50.0, dHL := 150.0, strAI := ai.T_masla_posle_AVOM);
  inits := inits + BOOL_TO_UINT(stAI_Ini.Init);

  (* [A1-6, AI2-6] Т газа на входе нагнетателя *)
  stAI_Ini(data_Ini := TRUE,  dLL := -50.0, dHL := 150.0, strAI := ai.T_gaz_in_nagnetatelia);
  inits := inits + BOOL_TO_UINT(stAI_Ini.Init);

  (* [A1-6, AI2-7]  Т газа на выходе нагнетателя *)
  stAI_Ini(data_Ini := TRUE,  dLL := -50.0, dHL := 150.0,
  ISVALIDREF_HA := TRUE, ISVALIDREF_HW := TRUE, dHA := 80.0, dHW := 60.0,
  strAI := ai.T_gaz_out_nagnetatelia);
  inits := inits + BOOL_TO_UINT(stAI_Ini.Init);

  (********************************************** Модуль A1-7 *********************************************************)
  (* [A1-7, AI3-0] Т горячего воздуха двигателя т.1 *)
  stAI_Ini(data_Ini := TRUE,  dLL := -50.0, dHL := 120.0, strAI := ai.T_hotAir_dvigatelia_t1);
  inits := inits + BOOL_TO_UINT(stAI_Ini.Init);

  (* [A1-7, AI3-2] Т холодного воздуха двигателя, т.1 *)
  stAI_Ini(data_Ini := TRUE,  dLL := -50.0, dHL := 120.0, strAI := ai.T_clodAir_dvigatelia_t1);
  inits := inits + BOOL_TO_UINT(stAI_Ini.Init);

  (********************************************** Модуль A1-8 *********************************************************)
  (* [A1-8, AI4-0]  Перепад давления "масло-газ" *)
  stAI_Ini(data_Ini := TRUE,  dLL := 0.0, dHL := 630.0,
  ISVALIDREF_LA := TRUE, ISVALIDREF_LW := TRUE, dLA := 100.0, dLW := 100.0, delayLA:=T#20S, delayLW:=T#4S,
  strAI := ai.dPmaslo_gaz);
  inits := inits + BOOL_TO_UINT(stAI_Ini.Init);

  (* [A1-8, AI4-1] Перепад давления газа на  конфузоре нагнетателя *)
  stAI_Ini(data_Ini := TRUE,  dLL := 0.0, dHL := 160.0, strAI := ai.dP_gaza_na_konfuzore_nagnetatelia);
  inits := inits + BOOL_TO_UINT(stAI_Ini.Init);

  (* [A1-8, AI4-2] Давление масла уплотнения *)
  stAI_Ini(data_Ini := TRUE,  dLL := 0.0, dHL := 10.0, strAI := ai.P_masla_uplotneniia);
  inits := inits + BOOL_TO_UINT(stAI_Ini.Init);

  (* [A1-8, AI4-3] Давление газа на входе нагнетателя *)
  stAI_Ini(data_Ini := TRUE,  dLL := 0.0, dHL := 10.0, strAI := ai.P_gaza_na_vkhode_nagnetatelia);
  inits := inits + BOOL_TO_UINT(stAI_Ini.Init);

  (* [A1-8, AI4-4] Давление газа на выходе нагнетателя *)
  stAI_Ini(data_Ini := TRUE,  dLL := 0.0, dHL := 10.0, strAI := ai.P_gaza_na_vykhode_nagnetatelia);
  inits := inits + BOOL_TO_UINT(stAI_Ini.Init);

  (* [A1-8, AI4-5]  Давление масла смазки низкое *)
  stAI_Ini(data_Ini := TRUE,  dLL := 0.0, dHL := 400.0,
  ISVALIDREF_LA := TRUE, ISVALIDREF_LW := TRUE, dLA := 40.0, dLW := 40.0, delayLA:=T#10S, delayLW:=T#4S,
  strAI := ai.P_masla_smazki_nizkoe);
  inits := inits + BOOL_TO_UINT(stAI_Ini.Init);

  (* [A1-8, AI4-6]  Давление масла смазки среднее (после насосов) *)
  stAI_Ini(data_Ini := TRUE,  dLL := 0.0, dHL := 1.0,
  ISVALIDREF_LW := TRUE, dLW := 0.4,
  strAI := ai.P_masla_smazki_srednee_posle_nasosov);
  inits := inits + BOOL_TO_UINT(stAI_Ini.Init);

  (********************************************** Модуль A1-9 *********************************************************)
  (* [A1-9, AI5-0]  Вибрация СТД т.1 *)
  stAI_Ini(data_Ini := TRUE,  dLL := 0.0, dHL := 20.0,
  ISVALIDREF_HA := TRUE, ISVALIDREF_HW := TRUE, dHA := 11.2, dHW := 4.5, aperturFilter:=0.05,
  strAI := ai.Vibratciia_STD_t1);
  inits := inits + BOOL_TO_UINT(stAI_Ini.Init);

  (* [A1-9, AI5-1]  Вибрация СТД т.2 *)
  stAI_Ini(data_Ini := TRUE,  dLL := 0.0, dHL := 20.0,
  ISVALIDREF_HA := TRUE, ISVALIDREF_HW := TRUE, dHA := 11.2, dHW := 4.5, aperturFilter:=0.05,
  strAI := ai.Vibratciia_STD_t2);
  inits := inits + BOOL_TO_UINT(stAI_Ini.Init);

  (* [A1-9, AI5-2]  Вибрация ротора нагнетателя т.1 *)
  stAI_Ini(data_Ini := TRUE,  dLL := 0.0, dHL := 250.0,
  ISVALIDREF_HA := TRUE, ISVALIDREF_HW := TRUE, dHA := 150.0, dHW := 125.0, aperturFilter:=0.05,
  strAI := ai.Vibratciia_rotora_nagnetatelia_t1);
  inits := inits + BOOL_TO_UINT(stAI_Ini.Init);

  (* [A1-9, AI5-3]  Вибрация ротора нагнетателя т.2 *)
  stAI_Ini(data_Ini := TRUE,  dLL := 0.0, dHL := 250.0,
  ISVALIDREF_HA := TRUE, ISVALIDREF_HW := TRUE, dHA := 150.0, dHW := 125.0, aperturFilter:=0.05,
  strAI := ai.Vibratciia_rotora_nagnetatelia_t2);
  inits := inits + BOOL_TO_UINT(stAI_Ini.Init);

  (* [A1-9, AI5-4]  Вибрация ротора нагнетателя т.3 *)
  stAI_Ini(data_Ini := TRUE,  dLL := 0.0, dHL := 250.0,
  ISVALIDREF_HA := TRUE, ISVALIDREF_HW := TRUE, dHA := 150.0, dHW := 125.0, aperturFilter:=0.05,
  strAI := ai.Vibratciia_rotora_nagnetatelia_t3);
  inits := inits + BOOL_TO_UINT(stAI_Ini.Init);

  (* [A1-9, AI5-5]  Вибрация ротора нагнетателя т.4 *)
  stAI_Ini(data_Ini := TRUE,  dLL := 0.0, dHL := 250.0,
  ISVALIDREF_HA := TRUE, ISVALIDREF_HW := TRUE, dHA := 150.0, dHW := 125.0, aperturFilter:=0.05,
  strAI := ai.Vibratciia_rotora_nagnetatelia_t4);
  inits := inits + BOOL_TO_UINT(stAI_Ini.Init);

  (* [A1-9, AI5-6]  Осевой сдвиг ротора нагнетателя *)
  stAI_Ini(data_Ini := TRUE,  dLL := -1.0, dHL := 1.0,
  ISVALIDREF_LA := TRUE, ISVALIDREF_HA := TRUE, ISVALIDREF_LW := TRUE, ISVALIDREF_HW := TRUE,
  dLA := -0.8, dHA := 0.8, dLW := -0.6, dHW := 0.6,
  strAI := ai.Osevoi_sdvig_rotora_nagnetatelia);
  inits := inits + BOOL_TO_UINT(stAI_Ini.Init);

  (* [A1-9, AI5-7]  Уровень масла в маслобаке *)
  stAI_Ini(data_Ini := TRUE,  dLL := 0.0, dHL := 1000.0,
  ISVALIDREF_LA := TRUE, ISVALIDREF_LW := TRUE, ISVALIDREF_HW := TRUE,
  dLA := 610.0, dLW := 670.0, dHW := 830.0,
  strAI := ai.Uroven_masla_v_maslobake);
  inits := inits + BOOL_TO_UINT(stAI_Ini.Init);

  (********************************************** Модуль A1-10 *********************************************************)

  (* [A1-10, AI6-0] Температура внутри шкафа *)
  stAI_Ini(data_Ini := TRUE,  dLL := -40.0, dHL := 80.0,
  ISVALIDREF_LW := TRUE, ISVALIDREF_HW := TRUE,
  dLW := 5.0, dHW := 50.0,
  strAI := ai.T_vnytri_shkafa);
  inits := inits + BOOL_TO_UINT(stAI_Ini.Init);

  (* [A1-10, AI6-2] Ток возбуждения возбудителя *)
  stAI_Ini(data_Ini := TRUE,  dLL := 0.0, dHL := 600.0, strAI := ai.Tok_vozbuzhdeniia_vozbuditelia);
  inits := inits + BOOL_TO_UINT(stAI_Ini.Init);

  (* [A1-10, AI6-3] Ток статора электродвигателя *)
  stAI_Ini(data_Ini := TRUE,  dLL := 0.0, dHL := 5.0, strAI := ai.Tok_statora_elektrodvigatelia);
  inits := inits + BOOL_TO_UINT(stAI_Ini.Init);

  (* [A1-10, AI6-4] Активная мощность *)
  stAI_Ini(data_Ini := TRUE,  dLL := 0.0, dHL := 15.0, strAI := ai.Aktivnaia_moshchnost);
  inits := inits + BOOL_TO_UINT(stAI_Ini.Init);

  (* [A1-10, AI6-5] Реактивная мощность *)
  stAI_Ini(data_Ini := TRUE,  dLL := 0.0, dHL := 15.0, strAI := ai.Reaktivnaia_moshchnost);
  inits := inits + BOOL_TO_UINT(stAI_Ini.Init);

  (* [A1-10, AI6-6]  Напряжение питания ШУ, основной ввод *)
  stAI_Ini(data_Ini := TRUE,  dLL := 0.0, dHL := 300.0,
  ISVALIDREF_LW := TRUE, ISVALIDREF_HW := TRUE, dLW := 187.0, dHW := 244.0,
  strAI := ai.VoltageSHU_osnovnoi_vvod);
  inits := inits + BOOL_TO_UINT(stAI_Ini.Init);

  (* [A1-10, AI6-7]  Напряжение питания ШУ, резервный ввод *)
  stAI_Ini(data_Ini := TRUE,  dLL := 0.0, dHL := 300.0,
  ISVALIDREF_LW := TRUE, ISVALIDREF_HW := TRUE, dLW := 187.0, dHW := 244.0,
  strAI := ai.VoltageSHU_rezervnyi_vvod);
  inits := inits + BOOL_TO_UINT(stAI_Ini.Init);

  initiales := 0;
  IF init THEN initiales := inits; END_IF;
END_FUNCTION_BLOCK

FUNCTION_BLOCK fb_sunpackerCommand
  VAR_INPUT
    command : WORD;
  END_VAR
  VAR_OUTPUT
    source : BYTE;
    parametr : BYTE;
    cmd : BYTE;
  END_VAR

  cmd := WORD_TO_BYTE(command and 16#7);
  parametr := WORD_TO_BYTE(SHR((command and 16#1FF8), 3));
  source := WORD_TO_BYTE(SHR(command, 13));
END_FUNCTION_BLOCK

FUNCTION_BLOCK fb_AiSourceMlp
  VAR_INPUT
    arAIN : TItemAIN;
    err_mod : TItemDIN;
  END_VAR
  VAR_IN_OUT
    strAI : struct_AI;
  END_VAR
  VAR
    _statusAi : TYPE_StatusAi;
    _commandAnalog : TYPE_CommandAnalog;
    _sunpackerCommand : fb_sunpackerCommand;
    _AnalogLimitFlags : TYPE_AnalogLimitFlags;
    notReliable : BOOL;
    _lastValue : LREAL;
    resetCmdTimer : TON;
    _LastValueTimer : TON;
    resetCmdTimerPriznak : BOOL;
    k : LREAL;
    b : LREAL;
    ap : LREAL;
    raznitsa : LREAL;
    rABS : LREAL;
    h : LREAL;
    mismatch : LREAL;
    parametr : BYTE;
    source : BYTE;
    cmd : BYTE;
    lastCmd : BYTE;
    source_for_Status : BYTE;
    cmd_for_Status : BYTE;
    command_error_for_Status : BYTE;
    onInit : BOOL;
    off_trig : R_TRIG;
    on_trig : R_TRIG;
    remont_trig : R_TRIG;
    LL_trig : R_TRIG;
    HL_trig : R_TRIG;
    Normal_trig : R_TRIG;
    Nedostover_trig : R_TRIG;
  END_VAR

  strAI.opcCommandsDisabled := strAI.inopcCommandsDisabled ;

  (* ---- При первом пуске принимаем значение уставок ---- *)
  IF NOT onInit THEN

            strAI.LL := strAI.dLL;
            strAI.HL := strAI.dHL;

            strAI.MaxChangeSpeed     := strAI.dMaxChangeSpeed;
            strAI.MaxChangeSpeedDown := strAI.dMaxChangeSpeedDown;

            IF strAI.ISVALIDREF_HA THEN strAI.HA := strAI.dHA; END_IF;

            IF strAI.ISVALIDREF_LA THEN strAI.LA := strAI.dLA; END_IF;

            IF strAI.ISVALIDREF_HW THEN strAI.HW := strAI.dHW; END_IF;

            IF strAI.ISVALIDREF_LW THEN strAI.LW := strAI.dLW; END_IF;

  	onInit  := TRUE;
  END_IF;

  (* ---- пересчет тока в физ величину ---- *)
  k := (strAI.HL - strAI.LL)/(strAI.inpHl - strAI.inpLL);
  b := strAI.LL - k * strAI.inpLL;
  strAI.value := k * arAIN.dblValue + b;

  (* ---- определение обрыва и кз ----- *)

  strAI.blConnect :=(*(UINT_TO_WORD(arAIN.wFlags) = 1472) and*) (UINT_TO_WORD(err_mod.wValue) = 20) and (UINT_TO_WORD(err_mod.wFlags) = 192);
  IF NOT strAI.blConnect THEN
      strAI.interval := _statusAi.NOTDEFINED;
  ELSIF ((arAIN.dblValue < strAI.currentBreakCircuit) AND (strAI.currentBreakCircuit > 0.0)) OR ((strAI.interval = _statusAi.LL) AND (arAIN.dblValue < (strAI.currentBreakCircuit + 100.0))) THEN
      strAI.interval := _statusAi.LL;
  ELSIF ((arAIN.dblValue > strAI.currentShotCircuit) AND (strAI.currentShotCircuit > 0.0)) OR ((strAI.interval = _statusAi.HL) AND (arAIN.dblValue > (strAI.currentShotCircuit - 100.0))) THEN
      strAI.interval := _statusAi.HL;
  ELSE
      strAI.interval := _statusAi.normal;
  END_IF;

  IF NOT strAI.imit THEN
  	(* Расчет апертурного фильтра*)
  	ap := strAI.aperturFilter * 0.01 * (strAI.HL - strAI.LL);
  	IF strAI.aperturFilter <> 0.0 THEN raznitsa := strAI.value- _lastValue;
  		IF 	raznitsa < 0.0 	THEN 	rABS := -raznitsa; 		ELSE 	rABS := raznitsa; 		END_IF;
  		IF 	rABS > ap 	THEN 	strAI.value := strAI.value;	ELSE 	strAI.value := _lastValue; 	END_IF;
  	END_IF;

  	(* Расчет экпоненциального фильтра*)
  	IF strAI.exponentialFilter <> 0.0 THEN strAI.value := (strAI.exponentialFilter * strAI.value) + ((1.0 - strAI.exponentialFilter) * _lastValue); END_IF;
  ELSE
  	strAI.interval := _statusAi.normal;
  END_IF;

  IF notReliable THEN strAI.interval := _statusAi.NOTRELIABLE; END_IF;

  IF NOT notReliable THEN
  	IF strAI.interval >= _statusAi.normal THEN
  		strAI.interval := _statusAi.NOTDEFINED;
  		h := strAI.histeresis* 0.01 * (strAI.HL-strAI.LL);
  		(*определение выхода за аппаратные границы вынесено в GetData.здесь только для нужд имитации*)
  		IF strAI.imit THEN
  			mismatch := strAI.rassoglasovanie * 0.01 * (strAI.HL - strAI.LL);
  			IF ( strAI.value < strAI.LL - mismatch)   THEN strAI.interval := _statusAi.LL;
  			ELSIF  (strAI.value > strAI.Hl + mismatch) THEN strAI.interval := _statusAi.HL; END_IF;
  		ELSE
  			strAI.interval := _statusAi.normal;
  			IF strAI.ISVALIDREF_LA AND NOT strAI.Disabled_LA AND (strAI.interval = _statusAi.normal) THEN
  				IF (strAI.value  < strAI.LA) OR ((strAI.interval = _statusAi.LA)  AND ((strAI.value - h) < strAI.LA))  THEN
  					strAI.interval := _statusAi.LA;
  				END_IF;
  			END_IF;
  			IF strAI.ISVALIDREF_HA  AND NOT strAI.Disabled_HA AND (strAI.interval = _statusAi.normal)  THEN
  				IF (strAI.value > strAI.HA) OR ((strAI.interval = _statusAi.HA)  AND ((strAI.value + h) > strAI.HA))  THEN
  					strAI.interval := _statusAi.HA;
  				END_IF;
  			END_IF;
  			IF strAI.ISVALIDREF_LW AND NOT strAI.Disabled_LW AND (strAI.interval = _statusAi.normal)  THEN
  				IF (strAI.value < strAI.LW) OR ((strAI.interval = _statusAi.LW)  AND ((strAI.value - h) < strAI.LW)) THEN
  					strAI.interval := _statusAi.LW;
  				END_IF;
  			END_IF;
  			IF strAI.ISVALIDREF_HW AND NOT strAI.Disabled_HW  AND (strAI.interval = _statusAi.normal) THEN
  				IF (strAI.value > strAI.HW)  OR ((strAI.interval = _statusAi.HW)  AND ((strAI.value + h) > strAI.HW))   THEN
  					strAI.interval := _statusAi.HW;
  				END_IF;
  			END_IF;
  		END_IF;
  	END_IF;
  ELSE
  	strAI.interval := _statusAi.NOTRELIABLE;
  END_IF;

  IF strAI.remont THEN strAI.interval := _statusAi.NOTDEFINED; END_IF;

  (* ---- Если управление с ВУ заблокировано, то  передаем команду из алгоритма ---- *)
  IF strAI.inOpcCommandsDisabled THEN
  	strAI.inCommand := strAI.inCommand_Alg;
  ELSE (* иначе передаем команду с АРМа*)
  	strAI.inCommand := strAI.inCommand_ARM;
  END_IF;

  _sunpackerCommand(command := strAI.inCommand);
  	source := _sunpackerCommand.source;
  	parametr := _sunpackerCommand.parametr;
  	cmd := _sunpackerCommand.cmd;

  IF cmd <> 0 AND lastCmd <> cmd and (((NOT strAI.opcCommandsDisabled) AND source > 0) OR source = 0) then
  	CASE BYTE_TO_INT(cmd) OF
  	(*cmd_SetUstavki*) 1 :
  				IF ((parametr AND _AnalogLimitFlags.LL) <> 0)		             	THEN 	strAI.LL := strAI.dLL; END_IF;
  				IF ((parametr AND _AnalogLimitFlags.HL) <> 0)		 	          THEN	strAI.HL := strAI.dHL; END_IF;
  				IF ((parametr AND _AnalogLimitFlags.LA) <> 0) AND strAI.ISVALIDREF_LA 	THEN	strAI.LA := strAI.dLA; END_IF;
  				IF ((parametr AND _AnalogLimitFlags.HA) <> 0) AND strAI.ISVALIDREF_HA 	THEN	strAI.HA := strAI.dHA; END_IF;
  				IF ((parametr AND _AnalogLimitFlags.LW) <> 0) AND strAI.ISVALIDREF_LW 	THEN	strAI.LW := strAI.dLW; END_IF;
  				IF ((parametr AND _AnalogLimitFlags.HW) <> 0) AND strAI.ISVALIDREF_HW 	THEN	strAI.HW := strAI.dHW; END_IF;
                                          IF ((parametr AND _AnalogLimitFlags.SipUP) <> 0)                       	THEN	strAI.MaxChangeSpeed     := strAI.dMaxChangeSpeed;     END_IF;
  				IF ((parametr AND _AnalogLimitFlags.SipDown) <> 0)                      	THEN	strAI.MaxChangeSpeedDown := strAI.dMaxChangeSpeedDown; END_IF;

  	(*cmd_SetRemont*) 6 :
  				strAI.remont := TRUE;
  	(*cmd_ResetRemont*) 7 :
  				strAI.remont := FALSE;
  	(*cmd_kvitNotReliable*) 4 :
  				notReliable := FALSE;
  	END_CASE;
  	source_for_Status := source;
  	cmd_for_Status := cmd;
  	command_error_for_Status := 0;
  	resetCmdTimer(IN := FALSE);
  	resetCmdTimerPriznak := TRUE;
  END_IF;
  lastCmd := cmd;

  resetCmdTimer(IN := resetCmdTimerPriznak, PT := T#5S);
  IF resetCmdTimer.Q THEN
  	resetCmdTimerPriznak := FALSE;
  	source_for_Status := 0;
  	cmd_for_Status := 0;
  	command_error_for_Status := 0;
  END_IF;

  strAI.NS_Min := (strAI.value < strAI.minValue) AND strAI.minValue_ISVALIDREF;
  strAI.NS_Max := (strAI.value > strAI.maxValue) AND strAI.maxValue_ISVALIDREF;

  strAI.NS := (strAI.interval <= _statusAi.normal) AND NOT strAI.remont;

  Normal_trig(CLK := strAI.interval >= _statusAi.normal);

  IF NOT Normal_trig.Q THEN
  	_LastValueTimer(PT := T#1S);
  	IF (strAI.value<>_lastValue) OR _LastValueTimer.Q THEN
  		IF (_LastValueTimer.ET>T#0MS) THEN
  			strAI.ChangeSpeed:=(strAI.value-_lastValue)/(TIME_TO_LREAL(_LastValueTimer.ET));
  		END_IF;
  		_LastValueTimer(IN:=FALSE);

  		_LastValueTimer(IN:=TRUE);
  	END_IF;
  END_IF;
  _lastValue := strAI.value;

  IF ((strAI.maxChangeSpeed<>0.0) OR  (strAI.maxChangeSpeedDown<>0.0)) AND ( strAI.interval>=_statusAi.normal) THEN
  		IF (strAI.ChangeSpeed>0.0) THEN
  		    IF (strAI.ChangeSpeed > strAI.maxChangeSpeed) AND (strAI.maxChangeSpeed>0.0000001) THEN
  			 notReliable:=TRUE;
  		    END_IF;
  		ELSE
  		    IF (ABS(strAI.ChangeSpeed)>strAI.maxChangeSpeedDown) AND (strAI.maxChangeSpeedDown>0.0000001)  THEN
                                 notReliable:=TRUE;
  		    END_IF;
  		END_IF;

  END_IF;

  strAI.status := SHL(BYTE_TO_DWORD(source_for_Status), 29) 		              (* Источник команды *)
  			OR SHL(BYTE_TO_DWORD(cmd_for_Status), 26) 	    (* Команда *)
  			OR SHL(BYTE_TO_DWORD(command_error_for_Status), 23)   (* Ошибка команды *)
  			OR SHL(BOOL_TO_DWORD(strAI.OpcCommandsDisabled ), 21) (* Управление в ВУ заблокировано *)
  			OR SHL(BOOL_TO_DWORD(strAI.Disabled_HA), 9)		    (* ВА исключена из формирования интервала *)
  			OR SHL(BOOL_TO_DWORD(strAI.Disabled_LA), 8)		    (* НА исключена из формирования интервала *)
  			OR SHL(BOOL_TO_DWORD(strAI.Disabled_HW), 7)		    (* ВП исключена из формирования интервала *)
  			OR SHL(BOOL_TO_DWORD(strAI.Disabled_LW), 6)	              (* НП исключена из формирования интервала *)
  			OR SHL(BOOL_TO_DWORD(strAI.NS), 5)			    (* неиспарвность сигнала *)
  			OR SHL(BOOL_TO_DWORD(strAI.remont), 4)	              (* Выведен в ремонт *)
  			OR BYTE_TO_DWORD(strAI.interval);	              (* интервал *)
END_FUNCTION_BLOCK

FUNCTION_BLOCK fb_AiSourceMlp_timer
  VAR_INPUT
    arAIN : TItemAIN;
    err_mod : TItemDIN;
  END_VAR
  VAR_IN_OUT
    strAI : struct_AI;
  END_VAR
  VAR RETAIN
    retainLL : LREAL;
    retainHL : LREAL;
    retainLA : LREAL;
    retainHA : LREAL;
    retainLW : LREAL;
    retainHW : LREAL;
  END_VAR
  VAR
    _statusAi : TYPE_StatusAi;
    _commandAnalog : TYPE_CommandAnalog;
    _sunpackerCommand : fb_sunpackerCommand;
    _AnalogLimitFlags : TYPE_AnalogLimitFlags;
    notReliable : BOOL;
    _lastValue : LREAL;
    resetCmdTimer : TON;
    _LastValueTimer : TON;
    resetCmdTimerPriznak : BOOL;
    k : LREAL;
    b : LREAL;
    ap : LREAL;
    raznitsa : LREAL;
    rABS : LREAL;
    h : LREAL;
    mismatch : LREAL;
    parametr : BYTE;
    source : BYTE;
    cmd : BYTE;
    lastCmd : BYTE;
    source_for_Status : BYTE;
    cmd_for_Status : BYTE;
    command_error_for_Status : BYTE;
    secondTakt : BOOL;
    off_trig : R_TRIG;
    on_trig : R_TRIG;
    remont_trig : R_TRIG;
    LL_trig : R_TRIG;
    HL_trig : R_TRIG;
    Normal_trig : R_TRIG;
    Nedostover_trig : R_TRIG;
    timerLA : TON;
    timerHA : TON;
    timerLW : TON;
    timerHW : TON;
  END_VAR

  strAI.opcCommandsDisabled := strAI.inopcCommandsDisabled ;

  (* ---- При первом пуске принимаем значение уставок ---- *)
  IF NOT secondTakt THEN
            IF (strAI.dLL <> retainLL) AND (retainLL <> 0.0) THEN  strAI.LL := retainLL;
            ELSE strAI.LL := strAI.dLL; END_IF;
  	IF (strAI.dHL <> retainHL) AND (retainHL <> 0.0) THEN  strAI.HL := retainHL;
            ELSE strAI.HL := strAI.dHL; END_IF;

            IF strAI.ISVALIDREF_HA AND (strAI.dHA <> retainHA) AND (retainHA <> 0.0) THEN  strAI.HA := retainHA;
            ELSE strAI.HA := strAI.dHA; END_IF;

            IF strAI.ISVALIDREF_LA AND (strAI.dLA <> retainLA) AND (retainLA <> 0.0) THEN  strAI.LA := retainLA;
            ELSE strAI.LA := strAI.dLA; END_IF;

            IF strAI.ISVALIDREF_HW AND (strAI.dHW <> retainHW) AND (retainHW <> 0.0) THEN  strAI.HW := retainHW;
            ELSE strAI.HW := strAI.dHW; END_IF;

            IF strAI.ISVALIDREF_LW AND (strAI.dLW <> retainLW) AND (retainLW <> 0.0) THEN  strAI.LW := retainLW;
            ELSE strAI.LW := strAI.dLW; END_IF;

  	secondTakt  := TRUE;
  END_IF;

  (* ---- пересчет тока в физ величину ---- *)
  k := (strAI.HL - strAI.LL)/(strAI.inpHl - strAI.inpLL);
  b := strAI.LL - k * strAI.inpLL;
  strAI.value := k * arAIN.dblValue + b;

  (* ---- определение обрыва и кз ----- *)

  strAI.blConnect := true;(*(UINT_TO_WORD(arAIN.wFlags) = 1472) and (UINT_TO_WORD(err_mod.wValue) = 20) and (UINT_TO_WORD(err_mod.wFlags) = 192); *)
  IF NOT strAI.blConnect THEN
      strAI.interval := _statusAi.NOTDEFINED;
  ELSIF ((arAIN.dblValue < strAI.currentBreakCircuit) AND (strAI.currentBreakCircuit > 0.0)) OR ((strAI.interval = _statusAi.LL) AND (arAIN.dblValue < (strAI.currentBreakCircuit + 100.0))) THEN
      strAI.interval := _statusAi.LL;
  ELSIF ((arAIN.dblValue > strAI.currentShotCircuit) AND (strAI.currentShotCircuit > 0.0)) OR ((strAI.interval = _statusAi.HL) AND (arAIN.dblValue > (strAI.currentShotCircuit - 100.0))) THEN
      strAI.interval := _statusAi.HL;
  ELSE
      strAI.interval := _statusAi.normal;
  END_IF;

  IF NOT strAI.imit THEN
  	(* Расчет апертурного фильтра*)
  	ap := strAI.aperturFilter * 0.01 * (strAI.HL - strAI.LL);
  	IF strAI.aperturFilter <> 0.0 THEN raznitsa := strAI.value- _lastValue;
  		IF 	raznitsa < 0.0 	THEN 	rABS := -raznitsa; 		ELSE 	rABS := raznitsa; 		END_IF;
  		IF 	rABS > ap 	THEN 	strAI.value := strAI.value;	ELSE 	strAI.value := _lastValue; 	END_IF;
  	END_IF;

  	(* Расчет экпоненциального фильтра*)
  	IF strAI.exponentialFilter <> 0.0 THEN strAI.value := (strAI.exponentialFilter * strAI.value) + ((1.0 - strAI.exponentialFilter) * _lastValue); END_IF;
  ELSE
  	strAI.interval := _statusAi.normal;
  END_IF;

  IF notReliable THEN strAI.interval := _statusAi.NOTRELIABLE; END_IF;

  IF NOT notReliable THEN
  	IF strAI.interval >= _statusAi.normal THEN
  		strAI.interval := _statusAi.NOTDEFINED;
  		h := strAI.histeresis* 0.01 * (strAI.HL-strAI.LL);
  		(*определение выхода за аппаратные границы вынесено в GetData.здесь только для нужд имитации*)
  		IF strAI.imit THEN
  			mismatch := strAI.rassoglasovanie * 0.01 * (strAI.HL - strAI.LL);
  			IF ( strAI.value < strAI.LL - mismatch)   THEN strAI.interval := _statusAi.LL;
  			ELSIF  (strAI.value > strAI.Hl + mismatch) THEN strAI.interval := _statusAi.HL; END_IF;
  		ELSE
  			strAI.interval := _statusAi.normal;
  			IF strAI.ISVALIDREF_LA AND NOT strAI.Disabled_LA AND (strAI.interval = _statusAi.normal) THEN
                                timerLA(IN:=(strAI.value  < strAI.LA) OR ((strAI.interval = _statusAi.LA)  AND ((strAI.value - h) < strAI.LA)), PT:=strAI.delayLA);
  				IF timerLA.Q  THEN
  					strAI.interval := _statusAi.LA;
  				END_IF;
  			END_IF;
  			IF strAI.ISVALIDREF_HA  AND NOT strAI.Disabled_HA AND (strAI.interval = _statusAi.normal)  THEN
                                timerHA(IN:=(strAI.value > strAI.HA) OR ((strAI.interval = _statusAi.HA)  AND ((strAI.value + h) > strAI.HA)), PT:=strAI.delayHA);
  				IF timerHA.Q  THEN
  					strAI.interval := _statusAi.HA;
  				END_IF;
  			END_IF;
  			IF strAI.ISVALIDREF_LW AND NOT strAI.Disabled_LW AND (strAI.interval = _statusAi.normal)  THEN
                                timerLW(IN:=(strAI.value < strAI.LW) OR ((strAI.interval = _statusAi.LW)  AND ((strAI.value - h) < strAI.LW)), PT:=strAI.delayLW);
  				IF timerLW.Q THEN
  					strAI.interval := _statusAi.LW;
  				END_IF;
  			END_IF;
  			IF strAI.ISVALIDREF_HW AND NOT strAI.Disabled_HW  AND (strAI.interval = _statusAi.normal) THEN
                                timerHW(IN:=(strAI.value > strAI.HW)  OR ((strAI.interval = _statusAi.HW)  AND ((strAI.value + h) > strAI.HW)), PT:=strAI.delayHW);
  				IF  timerHW.Q  THEN
  					strAI.interval := _statusAi.HW;
  				END_IF;
  			END_IF;
  		END_IF;
  	END_IF;
  ELSE
  	strAI.interval := _statusAi.NOTRELIABLE;
  END_IF;

  IF strAI.remont THEN strAI.interval := _statusAi.NOTDEFINED; END_IF;

  _sunpackerCommand(command := strAI.inCommand);
  	source := _sunpackerCommand.source;
  	parametr := _sunpackerCommand.parametr;
  	cmd := _sunpackerCommand.cmd;

  IF cmd <> 0 AND lastCmd <> cmd and (((NOT strAI.opcCommandsDisabled) AND source > 0) OR source = 0) then
  	CASE BYTE_TO_INT(cmd) OF
  	(*cmd_SetUstavki*) 1 :
  				IF ((parametr AND _AnalogLimitFlags.LL) <> 0)		             	THEN 	strAI.LL := strAI.dLL; retainLL:= strAI.LL; END_IF;
  				IF ((parametr AND _AnalogLimitFlags.HL) <> 0)		 	          THEN	strAI.HL := strAI.dHL; retainHL:= strAI.HL; END_IF;
  				IF ((parametr AND _AnalogLimitFlags.LA) <> 0) AND strAI.ISVALIDREF_LA 	THEN	strAI.LA := strAI.dLA; retainLA:= strAI.LA; END_IF;
  				IF ((parametr AND _AnalogLimitFlags.HA) <> 0) AND strAI.ISVALIDREF_HA 	THEN	strAI.HA := strAI.dHA; retainHA:= strAI.HA; END_IF;
  				IF ((parametr AND _AnalogLimitFlags.LW) <> 0) AND strAI.ISVALIDREF_LW 	THEN	strAI.LW := strAI.dLW; retainLW:= strAI.LW; END_IF;
  				IF ((parametr AND _AnalogLimitFlags.HW) <> 0) AND strAI.ISVALIDREF_HW 	THEN	strAI.HW := strAI.dHW; retainHW:= strAI.HW; END_IF;
  	(*cmd_SetRemont*) 2 :
  				strAI.remont := TRUE;
  	(*cmd_ResetRemont*) 3 :
  				strAI.remont := FALSE;
  	(*cmd_kvitNotReliable*) 4 :
  				notReliable := FALSE;
  	END_CASE;
  	source_for_Status := source;
  	cmd_for_Status := cmd;
  	command_error_for_Status := 0;
  	resetCmdTimer(IN := FALSE);
  	resetCmdTimerPriznak := TRUE;
  END_IF;
  lastCmd := cmd;

  resetCmdTimer(IN := resetCmdTimerPriznak, PT := T#5S);
  IF resetCmdTimer.Q THEN
  	resetCmdTimerPriznak := FALSE;
  	source_for_Status := 0;
  	cmd_for_Status := 0;
  	command_error_for_Status := 0;
  END_IF;

  strAI.NS_Min := (strAI.value < strAI.minValue) AND strAI.minValue_ISVALIDREF;
  strAI.NS_Max := (strAI.value > strAI.maxValue) AND strAI.maxValue_ISVALIDREF;

  strAI.NS := (strAI.interval <= _statusAi.normal) AND NOT strAI.remont;

  Normal_trig(CLK := strAI.interval >= _statusAi.normal);

  IF NOT Normal_trig.Q THEN
  	_LastValueTimer(PT := T#1S);
  	IF (strAI.value<>_lastValue) OR _LastValueTimer.Q THEN
  		IF (_LastValueTimer.ET>T#0MS) THEN
  			strAI.ChangeSpeed:=(strAI.value-_lastValue)/(TIME_TO_LREAL(_LastValueTimer.ET)/1000.0);
  		END_IF;
  		_LastValueTimer(IN:=FALSE);

  		_LastValueTimer(IN:=TRUE);
  	END_IF;
  END_IF;
  _lastValue := strAI.value;

  IF ((strAI.maxChangeSpeed<>0.0) OR  (strAI.maxChangeSpeedDown<>0.0)) AND ( strAI.interval>=_statusAi.normal) THEN
  		IF (strAI.ChangeSpeed>0.0) THEN
  		    IF (strAI.ChangeSpeed > strAI.maxChangeSpeed) AND (strAI.maxChangeSpeed>0.0000001) THEN
  			 notReliable:=TRUE;
  		    END_IF;
  		ELSE
  		    IF (ABS(strAI.ChangeSpeed)>strAI.maxChangeSpeedDown) AND (strAI.maxChangeSpeedDown>0.0000001)  THEN
                                 notReliable:=TRUE;
  		    END_IF;
  		END_IF;

  END_IF;

  strAI.status := SHL(BYTE_TO_DWORD(source_for_Status), 29) 		              (* Источник команды *)
  			OR SHL(BYTE_TO_DWORD(cmd_for_Status), 26) 	    (* Команда *)
  			OR SHL(BYTE_TO_DWORD(command_error_for_Status), 23)   (* Ошибка команды *)
  			OR SHL(BOOL_TO_DWORD(strAI.OpcCommandsDisabled ), 21) (* Управление в ВУ заблокировано *)
  			OR SHL(BOOL_TO_DWORD(strAI.Disabled_HA), 9)		    (* ВА исключена из формирования интервала *)
  			OR SHL(BOOL_TO_DWORD(strAI.Disabled_LA), 8)		    (* НА исключена из формирования интервала *)
  			OR SHL(BOOL_TO_DWORD(strAI.Disabled_HW), 7)		    (* ВП исключена из формирования интервала *)
  			OR SHL(BOOL_TO_DWORD(strAI.Disabled_LW), 6)	              (* НП исключена из формирования интервала *)
  			OR SHL(BOOL_TO_DWORD(strAI.NS), 5)			    (* неиспарвность сигнала *)
  			OR SHL(BOOL_TO_DWORD(strAI.remont), 4)	              (* Выведен в ремонт *)
  			OR BYTE_TO_DWORD(strAI.interval);	              (* интервал *)
END_FUNCTION_BLOCK

FUNCTION_BLOCK proc_AI
  VAR
    fb_T_obmotki_fazy_1_k : fb_AiSourceMlp;
    fb_T_akt_zheleza_statora_1_k : fb_AiSourceMlp;
    fb_T_obmotki_fazy_2_k : fb_AiSourceMlp;
    fb_T_akt_zheleza_statora_2_k : fb_AiSourceMlp;
    fb_T_obmotki_fazy_3_k : fb_AiSourceMlp;
    fb_T_akt_zheleza_statora_3_k : fb_AiSourceMlp;
    fb_T_masla_v_maslobake : fb_AiSourceMlp;
    fb_T_per_opor_pod_dvigatelia_t1 : fb_AiSourceMlp;
    fb_T_zad_opor_pod_dvigatelia_t2 : fb_AiSourceMlp;
    fb_T_masla_na_slive_per_opor_pod_dvigatelia : fb_AiSourceMlp;
    fb_T_masla_na_slive_zad_opor_pod_dvigatelia : fb_AiSourceMlp;
    fb_T_podshipnika_reduktora_t1 : fb_AiSourceMlp;
    fb_T_podshipnika_reduktora_t2 : fb_AiSourceMlp;
    fb_T_podshipnika_reduktora_t3 : fb_AiSourceMlp;
    fb_T_podshipnika_reduktora_t4 : fb_AiSourceMlp;
    fb_T_opor_pod_nagnetatelia_t1 : fb_AiSourceMlp;
    fb_T_opor_pod_nagnetatelia_t2 : fb_AiSourceMlp;
    fb_T_opor_pod_nagnetatelia_t3 : fb_AiSourceMlp;
    fb_T_opor_upor_pod_nagnetatelia_t4 : fb_AiSourceMlp;
    fb_T_masla_do_AVOM : fb_AiSourceMlp;
    fb_T_masla_posle_AVOM : fb_AiSourceMlp;
    fb_T_gaz_in_nagnetatelia : fb_AiSourceMlp;
    fb_T_gaz_out_nagnetatelia : fb_AiSourceMlp;
    fb_T_hotAir_dvigatelia_t1 : fb_AiSourceMlp;
    fb_T_clodAir_dvigatelia_t1 : fb_AiSourceMlp;
    fb_dPmaslo_gaz : fb_AiSourceMlp_timer;
    fb_dP_gaza_na_konfuzore_nagnetatelia : fb_AiSourceMlp;
    fb_P_masla_uplotneniia : fb_AiSourceMlp;
    fb_P_gaza_na_vkhode_nagnetatelia : fb_AiSourceMlp;
    fb_P_gaza_na_vykhode_nagnetatelia : fb_AiSourceMlp;
    fb_P_masla_smazki_nizkoe : fb_AiSourceMlp_timer;
    fb_P_masla_smazki_srednee_posle_nasosov : fb_AiSourceMlp;
    fb_Vibratciia_STD_t1 : fb_AiSourceMlp;
    fb_Vibratciia_STD_t2 : fb_AiSourceMlp;
    fb_Vibratciia_rotora_nagnetatelia_t1 : fb_AiSourceMlp;
    fb_Vibratciia_rotora_nagnetatelia_t2 : fb_AiSourceMlp;
    fb_Vibratciia_rotora_nagnetatelia_t3 : fb_AiSourceMlp;
    fb_Vibratciia_rotora_nagnetatelia_t4 : fb_AiSourceMlp;
    fb_Osevoi_sdvig_rotora_nagnetatelia : fb_AiSourceMlp;
    fb_Uroven_masla_v_maslobake : fb_AiSourceMlp;
    fb_T_vnytri_shkafa : fb_AiSourceMlp;
    fb_Tok_vozbuzhdeniia_vozbuditelia : fb_AiSourceMlp;
    fb_Tok_statora_elektrodvigatelia : fb_AiSourceMlp;
    fb_Aktivnaia_moshchnost : fb_AiSourceMlp;
    fb_Reaktivnaia_moshchnost : fb_AiSourceMlp;
    fb_VoltageSHU_osnovnoi_vvod : fb_AiSourceMlp;
    fb_VoltageSHU_rezervnyi_vvod : fb_AiSourceMlp;
  END_VAR
  VAR_EXTERNAL
    arAIN_0 : TItemAIN;
    arAIN_1 : TItemAIN;
    arAIN_2 : TItemAIN;
    arAIN_3 : TItemAIN;
    arAIN_4 : TItemAIN;
    arAIN_5 : TItemAIN;
    arAIN_6 : TItemAIN;
    arAIN_7 : TItemAIN;
    arAIN_8 : TItemAIN;
    arAIN_9 : TItemAIN;
    arAIN_10 : TItemAIN;
    arAIN_11 : TItemAIN;
    arAIN_12 : TItemAIN;
    arAIN_13 : TItemAIN;
    arAIN_14 : TItemAIN;
    arAIN_15 : TItemAIN;
    ai : AiConfig;
    arAIN_16 : TItemAIN;
    arAIN_17 : TItemAIN;
    arAIN_18 : TItemAIN;
    arAIN_19 : TItemAIN;
    arAIN_20 : TItemAIN;
    arAIN_21 : TItemAIN;
    arAIN_22 : TItemAIN;
    arAIN_23 : TItemAIN;
    arAIN_24 : TItemAIN;
    arAIN_25 : TItemAIN;
    arAIN_26 : TItemAIN;
    arAIN_27 : TItemAIN;
    arAIN_28 : TItemAIN;
    arAIN_29 : TItemAIN;
    arAIN_30 : TItemAIN;
    arAIN_31 : TItemAIN;
    arAIN_32 : TItemAIN;
    arAIN_33 : TItemAIN;
    arAIN_34 : TItemAIN;
    arAIN_35 : TItemAIN;
    arAIN_36 : TItemAIN;
    arAIN_37 : TItemAIN;
    arAIN_38 : TItemAIN;
    arAIN_39 : TItemAIN;
    arAIN_40 : TItemAIN;
    arAIN_41 : TItemAIN;
    arAIN_42 : TItemAIN;
    arAIN_43 : TItemAIN;
    arAIN_44 : TItemAIN;
    arAIN_45 : TItemAIN;
    arAIN_46 : TItemAIN;
    arAIN_47 : TItemAIN;
    arAIN_48 : TItemAIN;
    arAIN_49 : TItemAIN;
    arAIN_50 : TItemAIN;
    arAIN_51 : TItemAIN;
    arAIN_52 : TItemAIN;
    arAIN_53 : TItemAIN;
    arAIN_54 : TItemAIN;
    arAIN_55 : TItemAIN;
    arERR_3 : TItemDIN;
    arERR_4 : TItemDIN;
    arERR_5 : TItemDIN;
    arERR_6 : TItemDIN;
    arERR_7 : TItemDIN;
    arERR_8 : TItemDIN;
    arERR_9 : TItemDIN;
    A1_10_err_mode : UINT;
    A1_11_err_mode : UINT;
    A1_4_err_mode : UINT;
    A1_5_err_mode : UINT;
    A1_6_err_mode : UINT;
    A1_7_err_mode : UINT;
    A1_8_err_mode : UINT;
    A1_9_err_mode : UINT;
    A2_2_err_mode : UINT;
    A2_3_err_mode : UINT;
    AI_0_dblValue : LREAL;
    AI_10_dblValue : LREAL;
    AI_11_dblValue : LREAL;
    AI_12_dblValue : LREAL;
    AI_13_dblValue : LREAL;
    AI_14_dblValue : LREAL;
    AI_15_dblValue : LREAL;
    AI_16_dblValue : LREAL;
    AI_17_dblValue : LREAL;
    AI_18_dblValue : LREAL;
    AI_19_dblValue : LREAL;
    AI_1_dblValue : LREAL;
    AI_20_dblValue : LREAL;
    AI_21_dblValue : LREAL;
    AI_22_dblValue : LREAL;
    AI_23_dblValue : LREAL;
    AI_24_dblValue : LREAL;
    AI_25_dblValue : LREAL;
    AI_26_dblValue : LREAL;
    AI_27_dblValue : LREAL;
    AI_28_dblValue : LREAL;
    AI_29_dblValue : LREAL;
    AI_2_dblValue : LREAL;
    AI_30_dblValue : LREAL;
    AI_31_dblValue : LREAL;
    AI_32_dblValue : LREAL;
    AI_33_dblValue : LREAL;
    AI_34_dblValue : LREAL;
    AI_35_dblValue : LREAL;
    AI_36_dblValue : LREAL;
    AI_37_dblValue : LREAL;
    AI_38_dblValue : LREAL;
    AI_39_dblValue : LREAL;
    AI_3_dblValue : LREAL;
    AI_40_dblValue : LREAL;
    AI_41_dblValue : LREAL;
    AI_42_dblValue : LREAL;
    AI_43_dblValue : LREAL;
    AI_44_dblValue : LREAL;
    AI_45_dblValue : LREAL;
    AI_46_dblValue : LREAL;
    AI_47_dblValue : LREAL;
    AI_48_dblValue : LREAL;
    AI_49_dblValue : LREAL;
    AI_4_dblValue : LREAL;
    AI_50_dblValue : LREAL;
    AI_51_dblValue : LREAL;
    AI_52_dblValue : LREAL;
    AI_53_dblValue : LREAL;
    AI_54_dblValue : LREAL;
    AI_55_dblValue : LREAL;
    AI_56_dblValue : LREAL;
    AI_57_dblValue : LREAL;
    AI_58_dblValue : LREAL;
    AI_59_dblValue : LREAL;
    AI_5_dblValue : LREAL;
    AI_60_dblValue : LREAL;
    AI_61_dblValue : LREAL;
    AI_62_dblValue : LREAL;
    AI_63_dblValue : LREAL;
    AI_64_dblValue : LREAL;
    AI_65_dblValue : LREAL;
    AI_66_dblValue : LREAL;
    AI_67_dblValue : LREAL;
    AI_68_dblValue : LREAL;
    AI_69_dblValue : LREAL;
    AI_6_dblValue : LREAL;
    AI_70_dblValue : LREAL;
    AI_71_dblValue : LREAL;
    AI_72_dblValue : LREAL;
    AI_73_dblValue : LREAL;
    AI_74_dblValue : LREAL;
    AI_75_dblValue : LREAL;
    AI_76_dblValue : LREAL;
    AI_77_dblValue : LREAL;
    AI_78_dblValue : LREAL;
    AI_79_dblValue : LREAL;
    AI_7_dblValue : LREAL;
    AI_8_dblValue : LREAL;
    AI_9_dblValue : LREAL;
  END_VAR

  (* Циклический опрос. Входные аналоговые параметры *)

  (********************************************* Модуль A1-4 ******************************************************)
  (* [A1-4, AI0-0] Т обмотки фазы 1 канал *)
  fb_T_obmotki_fazy_1_k(arAIN := arAIN_0, strAI := ai.T_obmotki_fazy_1_k, err_mod:=arERR_3);
  AI_0_dblValue := arAIN_0.dblValue;

  (* [A1-4, AI0-1] Т активного железа статора 1 канал *)
  fb_T_akt_zheleza_statora_1_k(arAIN := arAIN_1, strAI := ai.T_aktivnogo_zheleza_statora_1_k, err_mod:=arERR_3);
  AI_1_dblValue := arAIN_1.dblValue;

  (* [A1-4, AI0-2] ТТ обмотки фазы 2 канал *)
  fb_T_obmotki_fazy_2_k(arAIN := arAIN_2, strAI := ai.T_obmotki_fazy_2_k, err_mod:=arERR_3);
  AI_2_dblValue := arAIN_2.dblValue;

  (* [A1-4, AI0-3] Т активного железа статора 2 канал *)
  fb_T_akt_zheleza_statora_2_k(arAIN := arAIN_3, strAI := ai.T_aktivnogo_zheleza_statora_2_k, err_mod:=arERR_3);
  AI_3_dblValue := arAIN_3.dblValue;

  (* [A1-4, AI0-4] Т обмотки фазы 3 канал *)
  fb_T_obmotki_fazy_3_k(arAIN := arAIN_4, strAI := ai.T_obmotki_fazy_3_k, err_mod:=arERR_3);
  AI_4_dblValue := arAIN_4.dblValue;

  (* [A1-4, AI0-5] Т активного железа статора 3 канал *)
  fb_T_akt_zheleza_statora_3_k(arAIN := arAIN_5, strAI := ai.T_aktivnogo_zheleza_statora_3_k, err_mod:=arERR_3);
  AI_5_dblValue := arAIN_5.dblValue;

  (* [A1-4, AI0-6] Т масла в маслобаке } *)
  fb_T_masla_v_maslobake(arAIN := arAIN_6, strAI := ai.T_masla_v_maslobake, err_mod:=arERR_3);
  AI_6_dblValue := arAIN_6.dblValue;

  A1_4_err_mode := arERR_3.wValue;

  (********************************************** Модуль A1-5 *********************************************************)
  (* [A1-5, AI1-0]  Т переднего опорного подшипника двигателя, т.1 *)
  fb_T_per_opor_pod_dvigatelia_t1(arAIN := arAIN_8, strAI := ai.T_perednego_opornogo_podshipnika_dvigatelia_t1, err_mod:=arERR_4);
  AI_8_dblValue := arAIN_8.dblValue;

  (* [A1-5, AI1-1]  Т заднего опорного подшипника двигателя, т.2 *)
  fb_T_zad_opor_pod_dvigatelia_t2(arAIN := arAIN_9, strAI := ai.T_zadnego_opornogo_podshipnika_dvigatelia_t2, err_mod:=arERR_4);
  AI_9_dblValue := arAIN_9.dblValue;

  (* [A1-5, AI1-2] Т масла на сливе переднего опорного подшипника двигателя *)
  fb_T_masla_na_slive_per_opor_pod_dvigatelia(arAIN := arAIN_10, strAI := ai.T_masla_na_slive_perednego_opornogo_podshipnika_dvigatelia, err_mod:=arERR_4);
  AI_10_dblValue := arAIN_10.dblValue;

  (* [A1-5, AI1-3] Т масла на сливе заднего опорного подшипника двигателя *)
  fb_T_masla_na_slive_zad_opor_pod_dvigatelia(arAIN := arAIN_11, strAI := ai.T_masla_na_slive_zadnego_opornogo_podshipnika_dvigatelia, err_mod:=arERR_4);
  AI_11_dblValue := arAIN_11.dblValue;

  (* [A1-5, AI1-4]  Т подшипника редуктора, т1 *)
  fb_T_podshipnika_reduktora_t1(arAIN := arAIN_12, strAI := ai.T_podshipnika_reduktora_t1, err_mod:=arERR_4);
  AI_12_dblValue := arAIN_12.dblValue;

  (* [A1-5, AI1-5]  Т подшипника редуктора, т2 *)
  fb_T_podshipnika_reduktora_t2(arAIN := arAIN_13, strAI := ai.T_podshipnika_reduktora_t2, err_mod:=arERR_4);
  AI_13_dblValue := arAIN_13.dblValue;

  (* [A1-5, AI1-6]  Т подшипника редуктора, т3 *)
  fb_T_podshipnika_reduktora_t3(arAIN := arAIN_14, strAI := ai.T_podshipnika_reduktora_t3, err_mod:=arERR_4);
  AI_14_dblValue := arAIN_14.dblValue;

  (* [A1-5, AI1-7]  Т подшипника редуктора, т4 *)
  fb_T_podshipnika_reduktora_t4(arAIN := arAIN_15, strAI := ai.T_podshipnika_reduktora_t4, err_mod:=arERR_4);
  AI_15_dblValue := arAIN_15.dblValue;

  A1_5_err_mode := arERR_4.wValue;

  (********************************************** Модуль A1-6 *********************************************************)
  (* [A1-6, AI2-0]  Т опорного подшипника нагнетателя, т1 *)
  fb_T_opor_pod_nagnetatelia_t1(arAIN := arAIN_16, strAI := ai.T_opornogo_podshipnika_nagnetatelia_t1, err_mod:=arERR_5);
  AI_16_dblValue := arAIN_16.dblValue;

  (* [A1-6, AI2-1]  Т опорного подшипника нагнетателя, т2 *)
  fb_T_opor_pod_nagnetatelia_t2(arAIN := arAIN_17, strAI := ai.T_opornogo_podshipnika_nagnetatelia_t2, err_mod:=arERR_5);
  AI_17_dblValue := arAIN_17.dblValue;

  (* [A1-6, AI2-2]  Т опорного подшипника нагнетателя, т3 *)
  fb_T_opor_pod_nagnetatelia_t3(arAIN := arAIN_18, strAI := ai.T_opornogo_podshipnika_nagnetatelia_t3, err_mod:=arERR_5);
  AI_18_dblValue := arAIN_18.dblValue;

  (* [A1-6, AI2-3]  Т опорно-упорного подшипника нагнетателя, т4 *)
  fb_T_opor_upor_pod_nagnetatelia_t4(arAIN := arAIN_19, strAI := ai.T_oporno_upornogo_podshipnika_nagnetatelia_t4, err_mod:=arERR_5);
  AI_19_dblValue := arAIN_19.dblValue;

  (* [A1-6, AI2-4] Т масла до АВОМ *)
  fb_T_masla_do_AVOM(arAIN := arAIN_20, strAI := ai.T_masla_do_AVOM, err_mod:=arERR_5);
  AI_20_dblValue := arAIN_20.dblValue;

  (* [A1-6, AI2-5] Т масла после АВОМ *)
  fb_T_masla_posle_AVOM(arAIN := arAIN_21, strAI := ai.T_masla_posle_AVOM, err_mod:=arERR_5);
  AI_21_dblValue := arAIN_21.dblValue;

  (* [A1-6, AI2-6] Т газа на входе нагнетателя *)
  fb_T_gaz_in_nagnetatelia(arAIN := arAIN_22, strAI := ai.T_gaz_in_nagnetatelia, err_mod:=arERR_5);
  AI_22_dblValue := arAIN_22.dblValue;

  (* [A1-6, AI2-7]  Т газа на выходе нагнетателя *)
  fb_T_gaz_out_nagnetatelia(arAIN := arAIN_23, strAI := ai.T_gaz_out_nagnetatelia, err_mod:=arERR_5);
  AI_23_dblValue := arAIN_23.dblValue;

  A1_6_err_mode := arERR_5.wValue;

  (********************************************** Модуль A1-7 *********************************************************)
  (* [A1-7, AI3-0] Т горячего воздуха двигателя т.1 *)
  fb_T_hotAir_dvigatelia_t1(arAIN := arAIN_24, strAI := ai.T_hotAir_dvigatelia_t1, err_mod:=arERR_6);
  AI_24_dblValue := arAIN_24.dblValue;

  (* [A1-7, AI3-2] Т холодного воздуха двигателя, т.1 *)
  fb_T_clodAir_dvigatelia_t1(arAIN := arAIN_26, strAI := ai.T_clodAir_dvigatelia_t1, err_mod:=arERR_6);
  AI_26_dblValue := arAIN_26.dblValue;

  A1_7_err_mode := arERR_6.wValue;

  (********************************************** Модуль A1-8 *********************************************************)
  (* [A1-8, AI4-0]  Перепад давления "масло-газ" *)
  fb_dPmaslo_gaz(arAIN := arAIN_32, strAI := ai.dPmaslo_gaz, err_mod:=arERR_7);
  AI_32_dblValue := arAIN_32.dblValue;

  (* [A1-8, AI4-1] Перепад давления газа на  конфузоре нагнетателя *)
  fb_dP_gaza_na_konfuzore_nagnetatelia(arAIN := arAIN_33, strAI := ai.dP_gaza_na_konfuzore_nagnetatelia, err_mod:=arERR_7);
  AI_33_dblValue := arAIN_33.dblValue;

  (* [A1-8, AI4-2] Давление масла уплотнения *)
  fb_P_masla_uplotneniia(arAIN := arAIN_34, strAI := ai.P_masla_uplotneniia, err_mod:=arERR_7);
  AI_34_dblValue := arAIN_34.dblValue;

  (* [A1-8, AI4-3] Давление газа на входе нагнетателя *)
  fb_P_gaza_na_vkhode_nagnetatelia(arAIN := arAIN_35, strAI := ai.P_gaza_na_vkhode_nagnetatelia, err_mod:=arERR_7);
  AI_35_dblValue := arAIN_35.dblValue;

  (* [A1-8, AI4-4] Давление газа на выходе нагнетателя *)
  fb_P_gaza_na_vykhode_nagnetatelia(arAIN := arAIN_36, strAI := ai.P_gaza_na_vykhode_nagnetatelia, err_mod:=arERR_7);
  AI_36_dblValue := arAIN_36.dblValue;

  (* [A1-8, AI4-5]  Давление масла смазки низкое *)
  fb_P_masla_smazki_nizkoe(arAIN := arAIN_37, strAI := ai.P_masla_smazki_nizkoe, err_mod:=arERR_7);
  AI_37_dblValue := arAIN_37.dblValue;

  (* [A1-8, AI4-6]  Давление масла смазки среднее (после насосов) *)
  fb_P_masla_smazki_srednee_posle_nasosov(arAIN := arAIN_38, strAI := ai.P_masla_smazki_srednee_posle_nasosov, err_mod:=arERR_7);
  AI_38_dblValue := arAIN_38.dblValue;

  A1_8_err_mode := arERR_7.wValue;

  (********************************************** Модуль A1-9 *********************************************************)
  (* [A1-9, AI5-0]  Вибрация СТД т.1 *)
  fb_Vibratciia_STD_t1(arAIN := arAIN_40, strAI := ai.Vibratciia_STD_t1, err_mod:=arERR_8);
  AI_40_dblValue := arAIN_40.dblValue;

  (* [A1-9, AI5-1]  Вибрация СТД т.2 *)
  fb_Vibratciia_STD_t2(arAIN := arAIN_41, strAI := ai.Vibratciia_STD_t2, err_mod:=arERR_8);
  AI_41_dblValue := arAIN_41.dblValue;

  (* [A1-9, AI5-2]  Вибрация ротора нагнетателя т.1 *)
  fb_Vibratciia_rotora_nagnetatelia_t1(arAIN := arAIN_42, strAI := ai.Vibratciia_rotora_nagnetatelia_t1, err_mod:=arERR_8);
  AI_42_dblValue := arAIN_42.dblValue;

  (* [A1-9, AI5-3]  Вибрация ротора нагнетателя т.2 *)
  fb_Vibratciia_rotora_nagnetatelia_t2(arAIN := arAIN_43, strAI := ai.Vibratciia_rotora_nagnetatelia_t2, err_mod:=arERR_8);
  AI_43_dblValue := arAIN_43.dblValue;

  (* [A1-9, AI5-4]  Вибрация ротора нагнетателя т.3 *)
  fb_Vibratciia_rotora_nagnetatelia_t3(arAIN := arAIN_44, strAI := ai.Vibratciia_rotora_nagnetatelia_t3, err_mod:=arERR_8);
  AI_44_dblValue := arAIN_44.dblValue;

  (* [A1-9, AI5-5]  Вибрация ротора нагнетателя т.4 *)
  fb_Vibratciia_rotora_nagnetatelia_t4(arAIN := arAIN_45, strAI := ai.Vibratciia_rotora_nagnetatelia_t4, err_mod:=arERR_8);
  AI_45_dblValue := arAIN_45.dblValue;

  (* [A1-9, AI5-6]  Осевой сдвиг ротора нагнетателя *)
  fb_Osevoi_sdvig_rotora_nagnetatelia(arAIN := arAIN_46, strAI := ai.Osevoi_sdvig_rotora_nagnetatelia, err_mod:=arERR_8);
  AI_46_dblValue := arAIN_46.dblValue;

  (* [A1-9, AI5-7]  Уровень масла в маслобаке *)
  fb_Uroven_masla_v_maslobake(arAIN := arAIN_47, strAI := ai.Uroven_masla_v_maslobake, err_mod:=arERR_8);
  AI_47_dblValue := arAIN_47.dblValue;

  A1_9_err_mode := arERR_8.wValue;

  (********************************************** Модуль A1-10 *********************************************************)
  (* [A1-10, AI6-0] Температура внутри шкафа *)
  fb_T_vnytri_shkafa(arAIN := arAIN_48, strAI := ai.T_vnytri_shkafa, err_mod:=arERR_9);
  AI_48_dblValue := arAIN_48.dblValue;

  (* [A1-10, AI6-2] Ток возбуждения возбудителя *)
  fb_Tok_vozbuzhdeniia_vozbuditelia(arAIN := arAIN_50, strAI := ai.Tok_vozbuzhdeniia_vozbuditelia, err_mod:=arERR_9);
  AI_50_dblValue := arAIN_50.dblValue;

  (* [A1-10, AI6-3] Ток статора электродвигателя *)
  fb_Tok_statora_elektrodvigatelia(arAIN := arAIN_51, strAI := ai.Tok_statora_elektrodvigatelia, err_mod:=arERR_9);
  AI_51_dblValue := arAIN_51.dblValue;

  (* [A1-10, AI6-4] Активная мощность *)
  fb_Aktivnaia_moshchnost(arAIN := arAIN_52, strAI := ai.Aktivnaia_moshchnost, err_mod:=arERR_9);
  AI_52_dblValue := arAIN_52.dblValue;

  (* [A1-10, AI6-5] Реактивная мощность *)
  fb_Reaktivnaia_moshchnost(arAIN := arAIN_53, strAI := ai.Reaktivnaia_moshchnost, err_mod:=arERR_9);
  AI_53_dblValue := arAIN_53.dblValue;

  (* [A1-10, AI6-6]  Напряжение питания ШУ, основной ввод *)
  fb_VoltageSHU_osnovnoi_vvod(arAIN := arAIN_54, strAI := ai.VoltageSHU_osnovnoi_vvod, err_mod:=arERR_9);
  AI_54_dblValue := arAIN_54.dblValue;

  (* [A1-10, AI6-7]  Напряжение питания ШУ, резервный ввод *)
  fb_VoltageSHU_rezervnyi_vvod(arAIN := arAIN_55, strAI := ai.VoltageSHU_rezervnyi_vvod, err_mod:=arERR_9);
  AI_55_dblValue := arAIN_55.dblValue;

  A1_10_err_mode := arERR_9.wValue;
END_FUNCTION_BLOCK

FUNCTION_BLOCK fb_AO_Init
  VAR_INPUT
    data_Ini : BOOL;
    outLL : LREAL := 4000.0;
    outHL : LREAL := 20000.0;
    newLL : LREAL;
    newHL : LREAL;
    newLL_ISVALIDREF : BOOL;
    newHL_ISVALIDREF : BOOL;
  END_VAR
  VAR_IN_OUT
    strAO : struct_AO;
  END_VAR
  VAR_OUTPUT
    Init : BOOL := FALSE;
  END_VAR

  (*****            Функциональный блок переинициализации структуры-дескриптора канала аналогового ввода.            *****)

   Init := FALSE;

      IF data_Ini THEN                            (* Параметрам требуется переинициализация. *)
          strAO.outLL                := outLL;
          strAO.outHL                := outHL;
          strAO.newLL                := newLL;
          strAO.newHL                := newHL;
          strAO.newLL_ISVALIDREF     := newLL_ISVALIDREF;
          strAO.newHL_ISVALIDREF     := newHL_ISVALIDREF;
          data_Ini:=FALSE;
          Init := TRUE;
      END_IF;
   IF Init THEN
         (* outLL:=0.0;*)
         (* outHL:=0.0;*)
          newLL:=0.0;
          newHL:=0.0;
          newLL_ISVALIDREF:= FALSE;
          newHL_ISVALIDREF:= FALSE;
   END_IF;
END_FUNCTION_BLOCK

FUNCTION_BLOCK proc_AO_Init
  VAR_INPUT
    init : BOOL;
  END_VAR
  VAR
    stAO_Ini : fb_AO_Init;
    inits : UINT;
  END_VAR
  VAR_INPUT
    initiales : UINT;
  END_VAR
  VAR_EXTERNAL
    ao : AOConfig;
  END_VAR

  (* Инициализация начало. Входные аналоговые параметры *)

  inits := 0; (* Флаг необходимости инициализации структур-дескрипторов *)

  (* Модуль A10 *)
  (* [A10, AO0] Резерв (A) *)
  stAO_Ini(data_Ini := TRUE, (*outLL := 4000.0, outHL := 20000.0,*)
    newLL_ISVALIDREF := TRUE, newHL_ISVALIDREF := TRUE,
    newLL := 0.0, newHL := 100.0,
    strAO := ao.Reserv_AO_1);
  inits := inits + BOOL_TO_UINT(stAO_Ini.Init);

  (* [A1-10, AO1] Резерв (A) *)
  stAO_Ini(data_Ini := TRUE, (*outLL := 4000.0, outHL := 20000.0,*)
    (*newLL_ISVALIDREF := TRUE, newHL_ISVALIDREF := TRUE,*)
    (*newLL := 0.0, newHL := 100.0,*)
  strAO := ao.Reserv_AO_2);
  inits := inits + BOOL_TO_UINT(stAO_Ini.Init);

  initiales := 0;
  IF init THEN initiales := inits; END_IF;
END_FUNCTION_BLOCK

FUNCTION_BLOCK fb_AOSourceMlp
  VAR_IN_OUT
    OutCurrent : TDoubleData;
    strAO : struct_AO;
  END_VAR
  VAR_INPUT RETAIN
    retainLL : LREAL;
    retainHL : LREAL;
  END_VAR
  VAR
    _sunpackerCommand : fb_sunpackerCommand;
    source : BYTE;
    source_for_Status : BYTE;
    cmd : BYTE;
    cmd_for_Status : BYTE;
    lastCmd : BYTE;
    command_error_for_Status : BYTE;
    resetCmdTimer : TON;
    resetCmdTimerPriznak : BOOL;
    secondTack : BOOL;
    inOpcCommandsDisabled : BOOL;
  END_VAR

  IF NOT secondTack THEN
            IF (strAO.newLL <> retainLL) AND (retainLL <> 0.0) THEN  strAO.LL := retainLL;
            ELSE strAO.LL:= strAO.newLL; END_IF;
  	IF (strAO.newHL <> retainHL) AND (retainHL <> 0.0) THEN  strAO.HL := retainHL;
            ELSE strAO.HL:= strAO.newHL; END_IF;

  	secondTack  := FALSE;
  END_IF;
  strAO.blConnect :=(UINT_TO_WORD(OutCurrent.wFlags) AND 16#0040) <> 0;
  strAO.OpcCommandsDisabled := inOpcCommandsDisabled;

  _sunpackerCommand(command := strAO.inCommand);
  	source := _sunpackerCommand.source;
  	cmd := _sunpackerCommand.cmd;

  IF cmd <> 0 AND lastCmd <> cmd and (((NOT strAO.opcCommandsDisabled) AND source > 0) OR source = 0) then
  	CASE BYTE_TO_INT(cmd) OF
  	(*cmd_ChangeValue*) 1 : 	IF ((NOT strAO.newLL_ISVALIDREF) OR (strAO.nValue >= strAO.LL)) AND
                                             ((NOT strAO.newHL_ISVALIDREF) OR (strAO.nValue <= strAO.HL) ) THEN
  					strAO.Value := strAO.nValue;
  				END_IF;
  	(*cmd_ChangeLimits*) 2 : 	strAO.LL := strAO.newLL; retainLL:= strAO.LL;
  				strAO.HL := strAO.newHL; retainHL:= strAO.HL;
  	END_CASE;
  	source_for_Status := source;
  	cmd_for_Status := cmd;
  	command_error_for_Status := 0;
  	resetCmdTimer(IN := FALSE);
  	resetCmdTimerPriznak := TRUE;
  END_IF;
  lastCmd := cmd;

  IF (strAO.HL <> strAO.LL) THEN
  	OutCurrent.dblValue := ((strAO.Value - strAO.LL) * (strAO.outHL-strAO.outLL)/(strAO.HL - strAO.LL )) + strAO.outLL;
  END_IF;

  resetCmdTimer(IN := resetCmdTimerPriznak, PT := T#5S);
  IF resetCmdTimer.Q THEN
  	resetCmdTimerPriznak := FALSE;
  	source_for_Status := 0;
  	cmd_for_Status := 0;
  	command_error_for_Status := 0;
  END_IF;

  strAO.status := SHL(BYTE_TO_DWORD(source_for_Status), 29)
  			OR SHL(BYTE_TO_DWORD(cmd_for_Status), 26)
  			OR SHL(BYTE_TO_DWORD(command_error_for_Status), 23)
  			OR SHL(BOOL_TO_DWORD(strAO.OpcCommandsDisabled ), 21);
END_FUNCTION_BLOCK

FUNCTION_BLOCK proc_AO
  VAR
    fb_Reserv_AO_1 : fb_AOSourceMlp;
    fb_Reserv_AO_2 : fb_AOSourceMlp;
  END_VAR
  VAR_EXTERNAL
    ao : AOConfig;
    arAOUT_0 : TDoubleData;
    arAOUT_1 : TDoubleData;
  END_VAR

  (* Циклический опрос. Входные аналоговые параметры *)

  (* Модуль A10 *)

  (* [A10-1, AO0] Резерв (A10) *)
  fb_Reserv_AO_1(OutCurrent := arAOUT_0, strAO := ao.Reserv_AO_1);

  (* [A10-1, AO1] Резерв (A10) *)
  fb_Reserv_AO_2(OutCurrent := arAOUT_1, strAO := ao.Reserv_AO_2);
END_FUNCTION_BLOCK

FUNCTION_BLOCK fb_DI_Init
  VAR_INPUT
    data_Ini : BOOL;
    imit : BOOL := FALSE;
  END_VAR
  VAR_IN_OUT
    strDI : struct_DI;
  END_VAR
  VAR_OUTPUT
    Init : BOOL := FALSE;
  END_VAR

  (*****            Функциональный блок переинициализации структуры-дескриптора канала дискретного ввода        *****)

   Init := FALSE;

      IF data_Ini THEN                            (* Параметрам требуется переинициализация. *)
          strDI.imit       := imit;
          data_Ini:=FALSE;
          Init := TRUE;
      END_IF;
    IF Init THEN
  imit:=FALSE;
      END_IF;
END_FUNCTION_BLOCK

FUNCTION_BLOCK proc_DI_Init
  VAR_INPUT
    init : BOOL;
  END_VAR
  VAR
    stDI_Ini : fb_DI_Init;
    inits : UINT;
  END_VAR
  VAR_INPUT
    initiales : UINT;
  END_VAR
  VAR_EXTERNAL
    di : DiConfig;
  END_VAR

  (* Инициализация начало. Входные дискретные параметры *)

  inits := 0; (* Флаг необходимости инициализации структур-дескрипторов *)

  (* Модуль A1-1 *)

  stDI_Ini(data_Ini := true, imit:=FALSE, strDI := di.di_0);
  inits := inits + BOOL_TO_UINT(stDI_Ini.Init);

  stDI_Ini(data_Ini := true, imit:=FALSE, strDI := di.di_1);
  inits := inits + BOOL_TO_UINT(stDI_Ini.Init);

  (* Модуль A1-2 *)
  stDI_Ini(data_Ini := true, imit:=FALSE, strDI := di.di_2);
  inits := inits + BOOL_TO_UINT(stDI_Ini.Init);

  stDI_Ini(data_Ini := true, imit:=FALSE, strDI := di.di_3);
  inits := inits + BOOL_TO_UINT(stDI_Ini.Init);

  (* Модуль A1-3 *)
  stDI_Ini(data_Ini := true, imit:=FALSE, strDI := di.di_4);
  inits := inits + BOOL_TO_UINT(stDI_Ini.Init);

  stDI_Ini(data_Ini := true, imit:=FALSE, strDI := di.di_5);
  inits := inits + BOOL_TO_UINT(stDI_Ini.Init);

  (* Модуль A1-4 *)
  stDI_Ini(data_Ini := true, imit:=FALSE, strDI := di.di_6);
  inits := inits + BOOL_TO_UINT(stDI_Ini.Init);

  stDI_Ini(data_Ini := true, imit:=FALSE, strDI := di.di_7);
  inits := inits + BOOL_TO_UINT(stDI_Ini.Init);

  (* Модуль A1-5 *)
  stDI_Ini(data_Ini := true, imit:=FALSE,  strDI := di.di_8);
  inits := inits + BOOL_TO_UINT(stDI_Ini.Init);

  stDI_Ini(data_Ini := true, imit:=FALSE,  strDI := di.di_9);
  inits := inits + BOOL_TO_UINT(stDI_Ini.Init);

  (* Модуль A1-6 *)
  stDI_Ini(data_Ini := true, imit:=FALSE,  strDI := di.di_10);
  inits := inits + BOOL_TO_UINT(stDI_Ini.Init);

  stDI_Ini(data_Ini := true, imit:=FALSE,  strDI := di.di_11);
  inits := inits + BOOL_TO_UINT(stDI_Ini.Init);

  (* Модуль A1-7 *)
  stDI_Ini(data_Ini := true, imit:=FALSE, strDI := di.di_12);
  inits := inits + BOOL_TO_UINT(stDI_Ini.Init);

  stDI_Ini(data_Ini := true, imit:=FALSE, strDI := di.di_13);
  inits := inits + BOOL_TO_UINT(stDI_Ini.Init);

  (* Модуль A1-8 *)
  stDI_Ini(data_Ini := true, imit:=FALSE, strDI := di.di_14);
  inits := inits + BOOL_TO_UINT(stDI_Ini.Init);

  stDI_Ini(data_Ini := true, imit:=FALSE, strDI := di.di_15);
  inits := inits + BOOL_TO_UINT(stDI_Ini.Init);

  initiales := 0;
  IF init THEN initiales := inits; END_IF;
END_FUNCTION_BLOCK

FUNCTION_BLOCK fb_DiSourceMlp
  VAR_INPUT
    arDIN : TItemDIN;
    err_mod : TItemDIN;
  END_VAR
  VAR_IN_OUT
    strDI : struct_DI;
  END_VAR
  VAR_OUTPUT
    Bounce : BOOL;
  END_VAR
  VAR
    _value : WORD;
    _reliability : BOOL;
    bitNumber : INT;
    bitNum : INT;
  END_VAR

  strDI.blConnect := (*((UINT_TO_WORD(arDIN.wFlags) = 1472) and*) (UINT_TO_WORD(err_mod.wValue) = 20) and (UINT_TO_WORD(err_mod.wFlags) = 192);
  Bounce := (UINT_TO_WORD(arDIN.wFlags) AND 16#0020) <> 0;

  If NOT strDI.imit THEN
  _value:=UINT_TO_WORD(arDIN.wValue);

      IF strDI.blConnect THEN
            strDI.reliability:=0;
            strDI.value:=0;
  	FOR bitNumber:=0 TO 7 BY 1 DO

  		_reliability:=WORD_TO_BOOL(SHR(_value, bitNumber*2) AND 16#2);
  		strDI.reliability:=strDI.reliability OR SHL(BOOL_TO_WORD(_reliability),bitNumber);
  		IF _reliability THEN
  			strDI.value:=strDI.value OR SHL((SHR(_value, bitNumber*2) AND 16#1),bitNumber);
  		END_IF;
  	END_FOR;
      ELSE
  	strDI.reliability := 0;
      END_IF;

      FOR bitNum:=0 TO 15 BY 1 DO
  	          strDI.bits[bitNum].reliability :=WORD_TO_BOOL(SHR(strDI.reliability, bitNum) AND 16#1);
  	IF strDI.bits[bitNum].reliability THEN
  		strDI.bits[bitNum].value :=WORD_TO_BOOL(SHR(strDI.value, bitNum) AND 16#1);
                      strDI.bits[bitNum]._inversed :=NOT strDI.bits[bitNum].value;
  	END_IF;
      END_FOR;

  END_IF;
END_FUNCTION_BLOCK

FUNCTION TwoUint_To_UDINT : UDINT
  VAR_INPUT
    val1 : UINT;
    val2 : UINT;
  END_VAR

  TwoUint_To_UDINT:= DWORD_TO_UDINT(UINT_TO_DWORD(val1) OR shl(UINT_TO_DWORD(val2), 16));
END_FUNCTION

FUNCTION_BLOCK proc_DI
  VAR
    di_0 : fb_DiSourceMlp;
    di_1 : fb_DiSourceMlp;
    di_2 : fb_DiSourceMlp;
    di_3 : fb_DiSourceMlp;
    di_4 : fb_DiSourceMlp;
    di_5 : fb_DiSourceMlp;
    di_6 : fb_DiSourceMlp;
    di_7 : fb_DiSourceMlp;
    di_8 : fb_DiSourceMlp;
    di_9 : fb_DiSourceMlp;
    di_10 : fb_DiSourceMlp;
    di_11 : fb_DiSourceMlp;
    di_12 : fb_DiSourceMlp;
    di_13 : fb_DiSourceMlp;
    di_14 : fb_DiSourceMlp;
    di_15 : fb_DiSourceMlp;
  END_VAR
  VAR_EXTERNAL
    arDIN_0 : TItemDIN;
    arDIN_1 : TItemDIN;
    arDIN_2 : TItemDIN;
    arDIN_3 : TItemDIN;
    arDIN_4 : TItemDIN;
    arDIN_5 : TItemDIN;
    arDIN_6 : TItemDIN;
    arDIN_7 : TItemDIN;
    arDIN_8 : TItemDIN;
    arDIN_9 : TItemDIN;
    arDIN_10 : TItemDIN;
    arDIN_11 : TItemDIN;
    arDIN_12 : TItemDIN;
    arDIN_13 : TItemDIN;
    arDIN_14 : TItemDIN;
    arDIN_15 : TItemDIN;
    di : DiConfig;
    DI_0_1_wValue : UDINT;
    DI_10_11_wValue : UDINT;
    DI_12_13_wValue : UDINT;
    DI_14_15_wValue : UDINT;
    DI_16_17_wValue : UDINT;
    DI_18_19_wValue : UDINT;
    DI_20_21_wValue : UDINT;
    DI_2_3_wValue : UDINT;
    DI_4_5_wValue : UDINT;
    DI_6_7_wValue : UDINT;
    DI_8_9_wValue : UDINT;
    A1_12_err_mode : UINT;
    A1_13_err_mode : UINT;
    A1_14_err_mode : UINT;
    A1_15_err_mode : UINT;
    A2_10_err_mode : UINT;
    A2_4_err_mode : UINT;
    A2_5_err_mode : UINT;
    A2_6_err_mode : UINT;
    A2_7_err_mode : UINT;
    A2_8_err_mode : UINT;
    A2_9_err_mode : UINT;
    arERR_11 : TItemDIN;
    arERR_12 : TItemDIN;
    arERR_13 : TItemDIN;
    arERR_14 : TItemDIN;
    arERR_18 : TItemDIN;
    arERR_19 : TItemDIN;
    arERR_20 : TItemDIN;
    arERR_21 : TItemDIN;
  END_VAR

  (* Циклический опрос. Входные дискретные параметры *)

  (* Модуль A1-12 *)
  di_0(arDIN := arDIN_0, strDI:=di.di_0, err_mod:=arERR_11);
  di_1(arDIN := arDIN_1, strDI:=di.di_1, err_mod:=arERR_11);
  DI_0_1_wValue:=TwoUint_To_UDINT(arDIN_0.wValue, arDIN_1.wValue);
  A1_12_err_mode:= arERR_11.wValue;

  (* Модуль A1-13 *)
  di_2(arDIN := arDIN_2, strDI:=di.di_2,  err_mod:=arERR_12);
  di_3(arDIN := arDIN_3, strDI:=di.di_3,  err_mod:=arERR_12);
  DI_2_3_wValue:=TwoUint_To_UDINT(arDIN_2.wValue, arDIN_3.wValue);
  A1_13_err_mode:= arERR_12.wValue;

  (* Модуль A1-14 *)
  di_4(arDIN := arDIN_4, strDI:=di.di_4,  err_mod:=arERR_13);
  di_5(arDIN := arDIN_5, strDI:=di.di_5,  err_mod:=arERR_13);
  DI_4_5_wValue:=TwoUint_To_UDINT(arDIN_4.wValue, arDIN_5.wValue);
  A1_14_err_mode:= arERR_13.wValue;

  (* Модуль A1-15 *)
  di_6(arDIN := arDIN_6, strDI:=di.di_6,  err_mod:=arERR_14);
  di_7(arDIN := arDIN_7, strDI:=di.di_7,  err_mod:=arERR_14);
  DI_6_7_wValue:=TwoUint_To_UDINT(arDIN_6.wValue, arDIN_7.wValue);
  A1_15_err_mode:= arERR_14.wValue;

  (* Модуль A2-4 *)
  di_8(arDIN := arDIN_8, strDI:=di.di_8,  err_mod:=arERR_18);
  di_9(arDIN := arDIN_9, strDI:=di.di_9,  err_mod:=arERR_18);
  DI_8_9_wValue:=TwoUint_To_UDINT(arDIN_8.wValue, arDIN_9.wValue);
  A2_4_err_mode:= arERR_18.wValue;

  (* Модуль A2-5 *)
  di_10(arDIN := arDIN_10, strDI:=di.di_10,  err_mod:=arERR_19);
  di_11(arDIN := arDIN_11, strDI:=di.di_11,  err_mod:=arERR_19);
  DI_10_11_wValue:=TwoUint_To_UDINT(arDIN_10.wValue, arDIN_11.wValue);
  A2_5_err_mode:= arERR_19.wValue;

  (* Модуль A2-6 *)
  di_12(arDIN := arDIN_12, strDI:=di.di_12,  err_mod:=arERR_20);
  di_13(arDIN := arDIN_13, strDI:=di.di_13,  err_mod:=arERR_20);
  DI_12_13_wValue:=TwoUint_To_UDINT(arDIN_12.wValue, arDIN_13.wValue);
  A2_6_err_mode:= arERR_20.wValue;

  (* Модуль A2-7 *)
  di_14(arDIN := arDIN_14, strDI:=di.di_14,  err_mod:=arERR_21);
  di_15(arDIN := arDIN_15, strDI:=di.di_15,  err_mod:=arERR_21);
  DI_14_15_wValue:=TwoUint_To_UDINT(arDIN_14.wValue, arDIN_15.wValue);
  A2_7_err_mode:= arERR_21.wValue;
END_FUNCTION_BLOCK

FUNCTION_BLOCK fb_DO_Init
  VAR_INPUT
    data_Ini : BOOL;
    imit : BOOL := FALSE;
  END_VAR
  VAR_IN_OUT
    strDO : struct_DO;
  END_VAR
  VAR_OUTPUT
    Init : BOOL := FALSE;
  END_VAR

  (*****            Функциональный блок переинициализации структуры-дескриптора канала дискретного ввода.            *****)
   Init := FALSE;

      IF data_Ini THEN                            (* Параметрам требуется переинициализация. *)
          strDO.imit       := imit;
          data_Ini:=FALSE;
          Init := TRUE;
      END_IF;
    IF Init THEN
  imit:=FALSE;
     END_IF;
END_FUNCTION_BLOCK

FUNCTION_BLOCK proc_DO_Init
  VAR_INPUT
    init : BOOL;
  END_VAR
  VAR
    stDO_Ini : fb_DO_Init;
    inits : UINT;
  END_VAR
  VAR_INPUT
    initiales : UINT;
  END_VAR
  VAR_EXTERNAL
    od : DOconfig;
  END_VAR

  (* Инициализация начало. Входные дискретные параметры *)

  inits := 0; (* Флаг необходимости инициализации структур-дескрипторов *)

  (* Модуль A1-15 *)
  stDO_Ini(data_Ini := true, imit:=FALSE, strDO := od.do_0);
  inits := inits + BOOL_TO_UINT(stDO_Ini.Init);

  (* Модуль A1-16 *)
  stDO_Ini(data_Ini := true, imit:=FALSE, strDO := od.do_1);
  inits := inits + BOOL_TO_UINT(stDO_Ini.Init);

  (* Модуль A1-17 *)
  stDO_Ini(data_Ini := true, imit:=FALSE, strDO := od.do_2);
  inits := inits + BOOL_TO_UINT(stDO_Ini.Init);

  (* Модуль A1-18 *)
  stDO_Ini(data_Ini := true, imit:=FALSE, strDO := od.do_3);
  inits := inits + BOOL_TO_UINT(stDO_Ini.Init);

  (* Модуль A1-19 *)
  stDO_Ini(data_Ini := true, imit:=FALSE, strDO := od.do_4);
  inits := inits + BOOL_TO_UINT(stDO_Ini.Init);

  (* Модуль A1-20 *)
  stDO_Ini(data_Ini := true, imit:=FALSE, strDO := od.do_5);
  inits := inits + BOOL_TO_UINT(stDO_Ini.Init);

  (* Модуль A1-21 *)
  stDO_Ini(data_Ini := true, imit:=FALSE, strDO := od.do_6);
  inits := inits + BOOL_TO_UINT(stDO_Ini.Init);

  (* Модуль A1-22 *)
  stDO_Ini(data_Ini := true, imit:=FALSE, strDO := od.do_7);
  inits := inits + BOOL_TO_UINT(stDO_Ini.Init);

  (* Модуль A1-23 *)
  stDO_Ini(data_Ini := true, imit:=FALSE, strDO := od.gpio_out);
  inits := inits + BOOL_TO_UINT(stDO_Ini.Init);
  initiales := 0;

  IF init THEN initiales := inits; END_IF;
END_FUNCTION_BLOCK

FUNCTION_BLOCK fb_DOSourceMlp
  VAR_IN_OUT
    arDout : TWordData;
  END_VAR
  VAR_INPUT
    err_mod : TItemDIN;
  END_VAR
  VAR_IN_OUT
    strDO : struct_DO;
  END_VAR
  VAR
    bitNumber : INT;
  END_VAR

  strDO.blConnect := ((UINT_TO_WORD(err_mod.wValue) = 20) and (UINT_TO_WORD(err_mod.wFlags) = 192));

  strDO.value:=0;

  FOR bitNumber:=0 TO 15 BY 1 DO
  	strDO.value:=strDO.value OR (SHL(BOOL_TO_WORD(strDO.bits[bitNumber]),bitNumber));
  END_FOR;

  IF NOT strDO.imit THEN
  	 arDout.wValue:= WORD_TO_UINT(strDO.value);
  END_IF;
END_FUNCTION_BLOCK

FUNCTION_BLOCK proc_DO
  VAR
    do_0 : fb_DOSourceMlp;
    do_1 : fb_DOSourceMlp;
    do_2 : fb_DOSourceMlp;
    do_3 : fb_DOSourceMlp;
    gpio_out : fb_DOSourceMlp;
  END_VAR
  VAR_EXTERNAL
    od : DOconfig;
    arDOUT_0 : TWordData;
    arDOUT_1 : TWordData;
    arDOUT_2 : TWordData;
    arDOUT_3 : TWordData;
    arERR_66 : TItemDIN;
    arDOUT_66 : TWordData;
    arERR_0 : TItemDIN;
    arERR_1 : TItemDIN;
    arERR_2 : TItemDIN;
    arERR_15 : TItemDIN;
    A1_1_err_mode : UINT;
    A1_2_err_mode : UINT;
    A1_3_err_mode : UINT;
    A2_1_err_mode : UINT;
    DO_0_wValue : UINT;
    DO_1_wValue : UINT;
    DO_2_wValue : UINT;
    DO_3_wValue : UINT;
  END_VAR

  (* Циклический опрос. Входные дискретные параметры *)

  (* Модуль A1-1 *)
  do_0(arDout := arDOUT_0, strDO := od.do_0, err_mod:=arERR_0);
  DO_0_wValue:=arDOUT_0.wValue;
  A1_1_err_mode:= arERR_0.wValue;

  (* Модуль A1-2 *)
  do_1(arDout := arDOUT_1, strDO := od.do_1, err_mod:=arERR_1);
  DO_1_wValue:=arDOUT_1.wValue;
  A1_2_err_mode:= arERR_1.wValue;

  (* Модуль A1-3 *)
  do_2(arDout := arDOUT_2, strDO := od.do_2, err_mod:=arERR_2);
  DO_2_wValue:=arDOUT_2.wValue;
  A1_3_err_mode:= arERR_2.wValue;

  (* Модуль A2-1 *)
  do_3(arDout := arDOUT_3, strDO := od.do_3, err_mod:=arERR_15);
  DO_3_wValue:=arDOUT_3.wValue;
  A2_1_err_mode:= arERR_15.wValue;

  gpio_out(arDout := arDOUT_66, strDO := od.gpio_out, err_mod:=arERR_66);
END_FUNCTION_BLOCK

FUNCTION_BLOCK OPC_AI_init
  VAR_EXTERNAL
    ai : AiConfig;
    AI_Aktivnaia_moshchnost_HL : LREAL;
    AI_Aktivnaia_moshchnost_LL : LREAL;
    AI_Aktivnaia_moshchnost_command : UINT;
    AI_Aktivnaia_moshchnost_newHL : LREAL;
    AI_Aktivnaia_moshchnost_newLL : LREAL;
    AI_Aktivnaia_moshchnost_status : UDINT;
    AI_Aktivnaia_moshchnost_value : LREAL;
    AI_Osevoi_sdvig_rotora_nagnetatelia_HA : LREAL;
    AI_Osevoi_sdvig_rotora_nagnetatelia_HL : LREAL;
    AI_Osevoi_sdvig_rotora_nagnetatelia_HW : LREAL;
    AI_Osevoi_sdvig_rotora_nagnetatelia_LA : LREAL;
    AI_Osevoi_sdvig_rotora_nagnetatelia_LL : LREAL;
    AI_Osevoi_sdvig_rotora_nagnetatelia_LW : LREAL;
    AI_Osevoi_sdvig_rotora_nagnetatelia_command : UINT;
    AI_Osevoi_sdvig_rotora_nagnetatelia_newHA : LREAL;
    AI_Osevoi_sdvig_rotora_nagnetatelia_newHL : LREAL;
    AI_Osevoi_sdvig_rotora_nagnetatelia_newHW : LREAL;
    AI_Osevoi_sdvig_rotora_nagnetatelia_newLA : LREAL;
    AI_Osevoi_sdvig_rotora_nagnetatelia_newLL : LREAL;
    AI_Osevoi_sdvig_rotora_nagnetatelia_newLW : LREAL;
    AI_Osevoi_sdvig_rotora_nagnetatelia_status : UDINT;
    AI_Osevoi_sdvig_rotora_nagnetatelia_value : LREAL;
    AI_P_gaza_na_vkhode_nagnetatelia_HL : LREAL;
    AI_P_gaza_na_vkhode_nagnetatelia_LL : LREAL;
    AI_P_gaza_na_vkhode_nagnetatelia_command : UINT;
    AI_P_gaza_na_vkhode_nagnetatelia_newHL : LREAL;
    AI_P_gaza_na_vkhode_nagnetatelia_newLL : LREAL;
    AI_P_gaza_na_vkhode_nagnetatelia_status : UDINT;
    AI_P_gaza_na_vkhode_nagnetatelia_value : LREAL;
    AI_P_gaza_na_vykhode_nagnetatelia_HL : LREAL;
    AI_P_gaza_na_vykhode_nagnetatelia_LL : LREAL;
    AI_P_gaza_na_vykhode_nagnetatelia_command : UINT;
    AI_P_gaza_na_vykhode_nagnetatelia_newHL : LREAL;
    AI_P_gaza_na_vykhode_nagnetatelia_newLL : LREAL;
    AI_P_gaza_na_vykhode_nagnetatelia_status : UDINT;
    AI_P_gaza_na_vykhode_nagnetatelia_value : LREAL;
    AI_P_masla_smazki_nizkoe_HL : LREAL;
    AI_P_masla_smazki_nizkoe_LA : LREAL;
    AI_P_masla_smazki_nizkoe_LL : LREAL;
    AI_P_masla_smazki_nizkoe_LW : LREAL;
    AI_P_masla_smazki_nizkoe_command : UINT;
    AI_P_masla_smazki_nizkoe_newHL : LREAL;
    AI_P_masla_smazki_nizkoe_newLA : LREAL;
    AI_P_masla_smazki_nizkoe_newLL : LREAL;
    AI_P_masla_smazki_nizkoe_newLW : LREAL;
    AI_P_masla_smazki_nizkoe_status : UDINT;
    AI_P_masla_smazki_nizkoe_value : LREAL;
    AI_P_masla_smazki_srednee_posle_nasosov_HL : LREAL;
    AI_P_masla_smazki_srednee_posle_nasosov_LL : LREAL;
    AI_P_masla_smazki_srednee_posle_nasosov_LW : LREAL;
    AI_P_masla_smazki_srednee_posle_nasosov_command : UINT;
    AI_P_masla_smazki_srednee_posle_nasosov_newHL : LREAL;
    AI_P_masla_smazki_srednee_posle_nasosov_newLL : LREAL;
    AI_P_masla_smazki_srednee_posle_nasosov_newLW : LREAL;
    AI_P_masla_smazki_srednee_posle_nasosov_status : UDINT;
    AI_P_masla_smazki_srednee_posle_nasosov_value : LREAL;
    AI_P_masla_uplotneniia_HL : LREAL;
    AI_P_masla_uplotneniia_LL : LREAL;
    AI_P_masla_uplotneniia_command : UINT;
    AI_P_masla_uplotneniia_newHL : LREAL;
    AI_P_masla_uplotneniia_newLL : LREAL;
    AI_P_masla_uplotneniia_status : UDINT;
    AI_P_masla_uplotneniia_value : LREAL;
    AI_Reaktivnaia_moshchnost_HL : LREAL;
    AI_Reaktivnaia_moshchnost_LL : LREAL;
    AI_Reaktivnaia_moshchnost_command : UINT;
    AI_Reaktivnaia_moshchnost_newHL : LREAL;
    AI_Reaktivnaia_moshchnost_newLL : LREAL;
    AI_Reaktivnaia_moshchnost_status : UDINT;
    AI_Reaktivnaia_moshchnost_value : LREAL;
    AI_T_aktivnogo_zheleza_statora_1_k_HL : LREAL;
    AI_T_aktivnogo_zheleza_statora_1_k_LL : LREAL;
    AI_T_aktivnogo_zheleza_statora_1_k_command : UINT;
    AI_T_aktivnogo_zheleza_statora_1_k_newHL : LREAL;
    AI_T_aktivnogo_zheleza_statora_1_k_newLL : LREAL;
    AI_T_aktivnogo_zheleza_statora_1_k_status : UDINT;
    AI_T_aktivnogo_zheleza_statora_1_k_value : LREAL;
    AI_T_aktivnogo_zheleza_statora_2_k_HL : LREAL;
    AI_T_aktivnogo_zheleza_statora_2_k_LL : LREAL;
    AI_T_aktivnogo_zheleza_statora_2_k_command : UINT;
    AI_T_aktivnogo_zheleza_statora_2_k_newHL : LREAL;
    AI_T_aktivnogo_zheleza_statora_2_k_newLL : LREAL;
    AI_T_aktivnogo_zheleza_statora_2_k_status : UDINT;
    AI_T_aktivnogo_zheleza_statora_2_k_value : LREAL;
    AI_T_aktivnogo_zheleza_statora_3_k_HL : LREAL;
    AI_T_aktivnogo_zheleza_statora_3_k_LL : LREAL;
    AI_T_aktivnogo_zheleza_statora_3_k_command : UINT;
    AI_T_aktivnogo_zheleza_statora_3_k_newHL : LREAL;
    AI_T_aktivnogo_zheleza_statora_3_k_newLL : LREAL;
    AI_T_aktivnogo_zheleza_statora_3_k_status : UDINT;
    AI_T_aktivnogo_zheleza_statora_3_k_value : LREAL;
    AI_T_clodAir_dvigatelia_t1_HL : LREAL;
    AI_T_clodAir_dvigatelia_t1_LL : LREAL;
    AI_T_clodAir_dvigatelia_t1_command : UINT;
    AI_T_clodAir_dvigatelia_t1_newHL : LREAL;
    AI_T_clodAir_dvigatelia_t1_newLL : LREAL;
    AI_T_clodAir_dvigatelia_t1_status : UDINT;
    AI_T_clodAir_dvigatelia_t1_value : LREAL;
    AI_T_gaz_in_nagnetatelia_HL : LREAL;
    AI_T_gaz_in_nagnetatelia_LL : LREAL;
    AI_T_gaz_in_nagnetatelia_command : UINT;
    AI_T_gaz_in_nagnetatelia_newHL : LREAL;
    AI_T_gaz_in_nagnetatelia_newLL : LREAL;
    AI_T_gaz_in_nagnetatelia_status : UDINT;
    AI_T_gaz_in_nagnetatelia_value : LREAL;
    AI_T_gaz_out_nagnetatelia_HL : LREAL;
    AI_T_gaz_out_nagnetatelia_LL : LREAL;
    AI_T_gaz_out_nagnetatelia_command : UINT;
    AI_T_gaz_out_nagnetatelia_newHL : LREAL;
    AI_T_gaz_out_nagnetatelia_newLL : LREAL;
    AI_T_gaz_out_nagnetatelia_status : UDINT;
    AI_T_gaz_out_nagnetatelia_value : LREAL;
    AI_T_hotAir_dvigatelia_t1_HL : LREAL;
    AI_T_hotAir_dvigatelia_t1_LL : LREAL;
    AI_T_hotAir_dvigatelia_t1_command : UINT;
    AI_T_hotAir_dvigatelia_t1_newHL : LREAL;
    AI_T_hotAir_dvigatelia_t1_newLL : LREAL;
    AI_T_hotAir_dvigatelia_t1_status : UDINT;
    AI_T_hotAir_dvigatelia_t1_value : LREAL;
    AI_T_masla_do_AVOM_HL : LREAL;
    AI_T_masla_do_AVOM_LL : LREAL;
    AI_T_masla_do_AVOM_command : UINT;
    AI_T_masla_do_AVOM_newHL : LREAL;
    AI_T_masla_do_AVOM_newLL : LREAL;
    AI_T_masla_do_AVOM_status : UDINT;
    AI_T_masla_do_AVOM_value : LREAL;
    AI_T_masla_na_slive_perednego_opornogo_podshipnika_dvigatelia_HL : LREAL;
    AI_T_masla_na_slive_perednego_opornogo_podshipnika_dvigatelia_LL : LREAL;
    AI_T_masla_na_slive_perednego_opornogo_podshipnika_dvigatelia_command : UINT;
    AI_T_masla_na_slive_perednego_opornogo_podshipnika_dvigatelia_newHL : LREAL;
    AI_T_masla_na_slive_perednego_opornogo_podshipnika_dvigatelia_newLL : LREAL;
    AI_T_masla_na_slive_perednego_opornogo_podshipnika_dvigatelia_status : UDINT;
    AI_T_masla_na_slive_perednego_opornogo_podshipnika_dvigatelia_value : LREAL;
    AI_T_masla_na_slive_zadnego_opornogo_podshipnika_dvigatelia_HL : LREAL;
    AI_T_masla_na_slive_zadnego_opornogo_podshipnika_dvigatelia_LL : LREAL;
    AI_T_masla_na_slive_zadnego_opornogo_podshipnika_dvigatelia_command : UINT;
    AI_T_masla_na_slive_zadnego_opornogo_podshipnika_dvigatelia_newHL : LREAL;
    AI_T_masla_na_slive_zadnego_opornogo_podshipnika_dvigatelia_newLL : LREAL;
    AI_T_masla_na_slive_zadnego_opornogo_podshipnika_dvigatelia_status : UDINT;
    AI_T_masla_na_slive_zadnego_opornogo_podshipnika_dvigatelia_value : LREAL;
    AI_T_masla_posle_AVOM_HL : LREAL;
    AI_T_masla_posle_AVOM_LL : LREAL;
    AI_T_masla_posle_AVOM_command : UINT;
    AI_T_masla_posle_AVOM_newHL : LREAL;
    AI_T_masla_posle_AVOM_newLL : LREAL;
    AI_T_masla_posle_AVOM_status : UDINT;
    AI_T_masla_posle_AVOM_value : LREAL;
    AI_T_masla_v_maslobake_HL : LREAL;
    AI_T_masla_v_maslobake_HW : LREAL;
    AI_T_masla_v_maslobake_LL : LREAL;
    AI_T_masla_v_maslobake_LW : LREAL;
    AI_T_masla_v_maslobake_command : UINT;
    AI_T_masla_v_maslobake_newHL : LREAL;
    AI_T_masla_v_maslobake_newHW : LREAL;
    AI_T_masla_v_maslobake_newLL : LREAL;
    AI_T_masla_v_maslobake_newLW : LREAL;
    AI_T_masla_v_maslobake_status : UDINT;
    AI_T_masla_v_maslobake_value : LREAL;
    AI_T_obmotki_fazy_1_k_HL : LREAL;
    AI_T_obmotki_fazy_1_k_LL : LREAL;
    AI_T_obmotki_fazy_1_k_command : UINT;
    AI_T_obmotki_fazy_1_k_newHL : LREAL;
    AI_T_obmotki_fazy_1_k_newLL : LREAL;
    AI_T_obmotki_fazy_1_k_status : UDINT;
    AI_T_obmotki_fazy_1_k_value : LREAL;
    AI_T_obmotki_fazy_2_k_HL : LREAL;
    AI_T_obmotki_fazy_2_k_LL : LREAL;
    AI_T_obmotki_fazy_2_k_command : UINT;
    AI_T_obmotki_fazy_2_k_newHL : LREAL;
    AI_T_obmotki_fazy_2_k_newLL : LREAL;
    AI_T_obmotki_fazy_2_k_status : UDINT;
    AI_T_obmotki_fazy_2_k_value : LREAL;
    AI_T_obmotki_fazy_3_k_HL : LREAL;
    AI_T_obmotki_fazy_3_k_LL : LREAL;
    AI_T_obmotki_fazy_3_k_command : UINT;
    AI_T_obmotki_fazy_3_k_newHL : LREAL;
    AI_T_obmotki_fazy_3_k_newLL : LREAL;
    AI_T_obmotki_fazy_3_k_status : UDINT;
    AI_T_obmotki_fazy_3_k_value : LREAL;
    AI_T_oporno_upornogo_podshipnika_nagnetatelia_t4_HA : LREAL;
    AI_T_oporno_upornogo_podshipnika_nagnetatelia_t4_HL : LREAL;
    AI_T_oporno_upornogo_podshipnika_nagnetatelia_t4_HW : LREAL;
    AI_T_oporno_upornogo_podshipnika_nagnetatelia_t4_LL : LREAL;
    AI_T_oporno_upornogo_podshipnika_nagnetatelia_t4_command : UINT;
    AI_T_oporno_upornogo_podshipnika_nagnetatelia_t4_newHA : LREAL;
    AI_T_oporno_upornogo_podshipnika_nagnetatelia_t4_newHL : LREAL;
    AI_T_oporno_upornogo_podshipnika_nagnetatelia_t4_newHW : LREAL;
    AI_T_oporno_upornogo_podshipnika_nagnetatelia_t4_newLL : LREAL;
    AI_T_oporno_upornogo_podshipnika_nagnetatelia_t4_status : UDINT;
    AI_T_oporno_upornogo_podshipnika_nagnetatelia_t4_value : LREAL;
    AI_T_opornogo_podshipnika_nagnetatelia_t1_HA : LREAL;
    AI_T_opornogo_podshipnika_nagnetatelia_t1_HL : LREAL;
    AI_T_opornogo_podshipnika_nagnetatelia_t1_HW : LREAL;
    AI_T_opornogo_podshipnika_nagnetatelia_t1_LL : LREAL;
    AI_T_opornogo_podshipnika_nagnetatelia_t1_command : UINT;
    AI_T_opornogo_podshipnika_nagnetatelia_t1_newHA : LREAL;
    AI_T_opornogo_podshipnika_nagnetatelia_t1_newHL : LREAL;
    AI_T_opornogo_podshipnika_nagnetatelia_t1_newHW : LREAL;
    AI_T_opornogo_podshipnika_nagnetatelia_t1_newLL : LREAL;
    AI_T_opornogo_podshipnika_nagnetatelia_t1_status : UDINT;
    AI_T_opornogo_podshipnika_nagnetatelia_t1_value : LREAL;
    AI_T_opornogo_podshipnika_nagnetatelia_t2_HA : LREAL;
    AI_T_opornogo_podshipnika_nagnetatelia_t2_HL : LREAL;
    AI_T_opornogo_podshipnika_nagnetatelia_t2_HW : LREAL;
    AI_T_opornogo_podshipnika_nagnetatelia_t2_LL : LREAL;
    AI_T_opornogo_podshipnika_nagnetatelia_t2_command : UINT;
    AI_T_opornogo_podshipnika_nagnetatelia_t2_newHA : LREAL;
    AI_T_opornogo_podshipnika_nagnetatelia_t2_newHL : LREAL;
    AI_T_opornogo_podshipnika_nagnetatelia_t2_newHW : LREAL;
    AI_T_opornogo_podshipnika_nagnetatelia_t2_newLL : LREAL;
    AI_T_opornogo_podshipnika_nagnetatelia_t2_status : UDINT;
    AI_T_opornogo_podshipnika_nagnetatelia_t2_value : LREAL;
    AI_T_opornogo_podshipnika_nagnetatelia_t3_HA : LREAL;
    AI_T_opornogo_podshipnika_nagnetatelia_t3_HL : LREAL;
    AI_T_opornogo_podshipnika_nagnetatelia_t3_HW : LREAL;
    AI_T_opornogo_podshipnika_nagnetatelia_t3_LL : LREAL;
    AI_T_opornogo_podshipnika_nagnetatelia_t3_command : UINT;
    AI_T_opornogo_podshipnika_nagnetatelia_t3_newHA : LREAL;
    AI_T_opornogo_podshipnika_nagnetatelia_t3_newHL : LREAL;
    AI_T_opornogo_podshipnika_nagnetatelia_t3_newHW : LREAL;
    AI_T_opornogo_podshipnika_nagnetatelia_t3_newLL : LREAL;
    AI_T_opornogo_podshipnika_nagnetatelia_t3_status : UDINT;
    AI_T_opornogo_podshipnika_nagnetatelia_t3_value : LREAL;
    AI_T_perednego_opornogo_podshipnika_dvigatelia_t1_HL : LREAL;
    AI_T_perednego_opornogo_podshipnika_dvigatelia_t1_LL : LREAL;
    AI_T_perednego_opornogo_podshipnika_dvigatelia_t1_command : UINT;
    AI_T_perednego_opornogo_podshipnika_dvigatelia_t1_newHL : LREAL;
    AI_T_perednego_opornogo_podshipnika_dvigatelia_t1_newLL : LREAL;
    AI_T_perednego_opornogo_podshipnika_dvigatelia_t1_status : UDINT;
    AI_T_perednego_opornogo_podshipnika_dvigatelia_t1_value : LREAL;
    AI_T_podshipnika_reduktora_t1_HA : LREAL;
    AI_T_podshipnika_reduktora_t1_HL : LREAL;
    AI_T_podshipnika_reduktora_t1_HW : LREAL;
    AI_T_podshipnika_reduktora_t1_LL : LREAL;
    AI_T_podshipnika_reduktora_t1_command : UINT;
    AI_T_podshipnika_reduktora_t1_newHA : LREAL;
    AI_T_podshipnika_reduktora_t1_newHL : LREAL;
    AI_T_podshipnika_reduktora_t1_newHW : LREAL;
    AI_T_podshipnika_reduktora_t1_newLL : LREAL;
    AI_T_podshipnika_reduktora_t1_status : UDINT;
    AI_T_podshipnika_reduktora_t1_value : LREAL;
    AI_T_podshipnika_reduktora_t2_HA : LREAL;
    AI_T_podshipnika_reduktora_t2_HL : LREAL;
    AI_T_podshipnika_reduktora_t2_HW : LREAL;
    AI_T_podshipnika_reduktora_t2_LL : LREAL;
    AI_T_podshipnika_reduktora_t2_command : UINT;
    AI_T_podshipnika_reduktora_t2_newHA : LREAL;
    AI_T_podshipnika_reduktora_t2_newHL : LREAL;
    AI_T_podshipnika_reduktora_t2_newHW : LREAL;
    AI_T_podshipnika_reduktora_t2_newLL : LREAL;
    AI_T_podshipnika_reduktora_t2_status : UDINT;
    AI_T_podshipnika_reduktora_t2_value : LREAL;
    AI_T_podshipnika_reduktora_t3_HA : LREAL;
    AI_T_podshipnika_reduktora_t3_HL : LREAL;
    AI_T_podshipnika_reduktora_t3_HW : LREAL;
    AI_T_podshipnika_reduktora_t3_LL : LREAL;
    AI_T_podshipnika_reduktora_t3_command : UINT;
    AI_T_podshipnika_reduktora_t3_newHA : LREAL;
    AI_T_podshipnika_reduktora_t3_newHL : LREAL;
    AI_T_podshipnika_reduktora_t3_newHW : LREAL;
    AI_T_podshipnika_reduktora_t3_newLL : LREAL;
    AI_T_podshipnika_reduktora_t3_status : UDINT;
    AI_T_podshipnika_reduktora_t3_value : LREAL;
    AI_T_podshipnika_reduktora_t4_HA : LREAL;
    AI_T_podshipnika_reduktora_t4_HL : LREAL;
    AI_T_podshipnika_reduktora_t4_HW : LREAL;
    AI_T_podshipnika_reduktora_t4_LL : LREAL;
    AI_T_podshipnika_reduktora_t4_command : UINT;
    AI_T_podshipnika_reduktora_t4_newHA : LREAL;
    AI_T_podshipnika_reduktora_t4_newHL : LREAL;
    AI_T_podshipnika_reduktora_t4_newHW : LREAL;
    AI_T_podshipnika_reduktora_t4_newLL : LREAL;
    AI_T_podshipnika_reduktora_t4_status : UDINT;
    AI_T_podshipnika_reduktora_t4_value : LREAL;
    AI_T_zadnego_opornogo_podshipnika_dvigatelia_t2_HA : LREAL;
    AI_T_zadnego_opornogo_podshipnika_dvigatelia_t2_HL : LREAL;
    AI_T_zadnego_opornogo_podshipnika_dvigatelia_t2_HW : LREAL;
    AI_T_zadnego_opornogo_podshipnika_dvigatelia_t2_LL : LREAL;
    AI_T_zadnego_opornogo_podshipnika_dvigatelia_t2_command : UINT;
    AI_T_zadnego_opornogo_podshipnika_dvigatelia_t2_newHA : LREAL;
    AI_T_zadnego_opornogo_podshipnika_dvigatelia_t2_newHL : LREAL;
    AI_T_zadnego_opornogo_podshipnika_dvigatelia_t2_newHW : LREAL;
    AI_T_zadnego_opornogo_podshipnika_dvigatelia_t2_newLL : LREAL;
    AI_T_zadnego_opornogo_podshipnika_dvigatelia_t2_status : UDINT;
    AI_T_zadnego_opornogo_podshipnika_dvigatelia_t2_value : LREAL;
    AI_Tok_statora_elektrodvigatelia_HL : LREAL;
    AI_Tok_statora_elektrodvigatelia_LL : LREAL;
    AI_Tok_statora_elektrodvigatelia_command : UINT;
    AI_Tok_statora_elektrodvigatelia_newHL : LREAL;
    AI_Tok_statora_elektrodvigatelia_newLL : LREAL;
    AI_Tok_statora_elektrodvigatelia_status : UDINT;
    AI_Tok_statora_elektrodvigatelia_value : LREAL;
    AI_Tok_vozbuzhdeniia_vozbuditelia_HL : LREAL;
    AI_Tok_vozbuzhdeniia_vozbuditelia_LL : LREAL;
    AI_Tok_vozbuzhdeniia_vozbuditelia_command : UINT;
    AI_Tok_vozbuzhdeniia_vozbuditelia_newHL : LREAL;
    AI_Tok_vozbuzhdeniia_vozbuditelia_newLL : LREAL;
    AI_Tok_vozbuzhdeniia_vozbuditelia_status : UDINT;
    AI_Tok_vozbuzhdeniia_vozbuditelia_value : LREAL;
    AI_Uroven_masla_v_maslobake_HL : LREAL;
    AI_Uroven_masla_v_maslobake_HW : LREAL;
    AI_Uroven_masla_v_maslobake_LA : LREAL;
    AI_Uroven_masla_v_maslobake_LL : LREAL;
    AI_Uroven_masla_v_maslobake_LW : LREAL;
    AI_Uroven_masla_v_maslobake_command : UINT;
    AI_Uroven_masla_v_maslobake_newHL : LREAL;
    AI_Uroven_masla_v_maslobake_newHW : LREAL;
    AI_Uroven_masla_v_maslobake_newLA : LREAL;
    AI_Uroven_masla_v_maslobake_newLL : LREAL;
    AI_Uroven_masla_v_maslobake_newLW : LREAL;
    AI_Uroven_masla_v_maslobake_status : UDINT;
    AI_Uroven_masla_v_maslobake_value : LREAL;
    AI_Vibratciia_STD_t1_HA : LREAL;
    AI_Vibratciia_STD_t1_HL : LREAL;
    AI_Vibratciia_STD_t1_HW : LREAL;
    AI_Vibratciia_STD_t1_LL : LREAL;
    AI_Vibratciia_STD_t1_command : UINT;
    AI_Vibratciia_STD_t1_newHA : LREAL;
    AI_Vibratciia_STD_t1_newHL : LREAL;
    AI_Vibratciia_STD_t1_newHW : LREAL;
    AI_Vibratciia_STD_t1_newLL : LREAL;
    AI_Vibratciia_STD_t1_status : UDINT;
    AI_Vibratciia_STD_t1_value : LREAL;
    AI_Vibratciia_STD_t2_HA : LREAL;
    AI_Vibratciia_STD_t2_HL : LREAL;
    AI_Vibratciia_STD_t2_HW : LREAL;
    AI_Vibratciia_STD_t2_LL : LREAL;
    AI_Vibratciia_STD_t2_command : UINT;
    AI_Vibratciia_STD_t2_newHA : LREAL;
    AI_Vibratciia_STD_t2_newHL : LREAL;
    AI_Vibratciia_STD_t2_newHW : LREAL;
    AI_Vibratciia_STD_t2_newLL : LREAL;
    AI_Vibratciia_STD_t2_status : UDINT;
    AI_Vibratciia_STD_t2_value : LREAL;
    AI_Vibratciia_rotora_nagnetatelia_t1_HA : LREAL;
    AI_Vibratciia_rotora_nagnetatelia_t1_HL : LREAL;
    AI_Vibratciia_rotora_nagnetatelia_t1_HW : LREAL;
    AI_Vibratciia_rotora_nagnetatelia_t1_LL : LREAL;
    AI_Vibratciia_rotora_nagnetatelia_t1_command : UINT;
    AI_Vibratciia_rotora_nagnetatelia_t1_newHA : LREAL;
    AI_Vibratciia_rotora_nagnetatelia_t1_newHL : LREAL;
    AI_Vibratciia_rotora_nagnetatelia_t1_newHW : LREAL;
    AI_Vibratciia_rotora_nagnetatelia_t1_newLL : LREAL;
    AI_Vibratciia_rotora_nagnetatelia_t1_status : UDINT;
    AI_Vibratciia_rotora_nagnetatelia_t1_value : LREAL;
    AI_Vibratciia_rotora_nagnetatelia_t2_HA : LREAL;
    AI_Vibratciia_rotora_nagnetatelia_t2_HL : LREAL;
    AI_Vibratciia_rotora_nagnetatelia_t2_HW : LREAL;
    AI_Vibratciia_rotora_nagnetatelia_t2_LL : LREAL;
    AI_Vibratciia_rotora_nagnetatelia_t2_command : UINT;
    AI_Vibratciia_rotora_nagnetatelia_t2_newHA : LREAL;
    AI_Vibratciia_rotora_nagnetatelia_t2_newHL : LREAL;
    AI_Vibratciia_rotora_nagnetatelia_t2_newHW : LREAL;
    AI_Vibratciia_rotora_nagnetatelia_t2_newLL : LREAL;
    AI_Vibratciia_rotora_nagnetatelia_t2_status : UDINT;
    AI_Vibratciia_rotora_nagnetatelia_t2_value : LREAL;
    AI_Vibratciia_rotora_nagnetatelia_t3_HA : LREAL;
    AI_Vibratciia_rotora_nagnetatelia_t3_HL : LREAL;
    AI_Vibratciia_rotora_nagnetatelia_t3_HW : LREAL;
    AI_Vibratciia_rotora_nagnetatelia_t3_LL : LREAL;
    AI_Vibratciia_rotora_nagnetatelia_t3_command : UINT;
    AI_Vibratciia_rotora_nagnetatelia_t3_newHA : LREAL;
    AI_Vibratciia_rotora_nagnetatelia_t3_newHL : LREAL;
    AI_Vibratciia_rotora_nagnetatelia_t3_newHW : LREAL;
    AI_Vibratciia_rotora_nagnetatelia_t3_newLL : LREAL;
    AI_Vibratciia_rotora_nagnetatelia_t3_status : UDINT;
    AI_Vibratciia_rotora_nagnetatelia_t3_value : LREAL;
    AI_Vibratciia_rotora_nagnetatelia_t4_HA : LREAL;
    AI_Vibratciia_rotora_nagnetatelia_t4_HL : LREAL;
    AI_Vibratciia_rotora_nagnetatelia_t4_HW : LREAL;
    AI_Vibratciia_rotora_nagnetatelia_t4_LL : LREAL;
    AI_Vibratciia_rotora_nagnetatelia_t4_command : UINT;
    AI_Vibratciia_rotora_nagnetatelia_t4_newHA : LREAL;
    AI_Vibratciia_rotora_nagnetatelia_t4_newHL : LREAL;
    AI_Vibratciia_rotora_nagnetatelia_t4_newHW : LREAL;
    AI_Vibratciia_rotora_nagnetatelia_t4_newLL : LREAL;
    AI_Vibratciia_rotora_nagnetatelia_t4_status : UDINT;
    AI_Vibratciia_rotora_nagnetatelia_t4_value : LREAL;
    AI_VoltageSHU_osnovnoi_vvod_HL : LREAL;
    AI_VoltageSHU_osnovnoi_vvod_HW : LREAL;
    AI_VoltageSHU_osnovnoi_vvod_LL : LREAL;
    AI_VoltageSHU_osnovnoi_vvod_LW : LREAL;
    AI_VoltageSHU_osnovnoi_vvod_command : UINT;
    AI_VoltageSHU_osnovnoi_vvod_newHL : LREAL;
    AI_VoltageSHU_osnovnoi_vvod_newHW : LREAL;
    AI_VoltageSHU_osnovnoi_vvod_newLL : LREAL;
    AI_VoltageSHU_osnovnoi_vvod_newLW : LREAL;
    AI_VoltageSHU_osnovnoi_vvod_status : UDINT;
    AI_VoltageSHU_osnovnoi_vvod_value : LREAL;
    AI_VoltageSHU_rezervnyi_vvod_HL : LREAL;
    AI_VoltageSHU_rezervnyi_vvod_HW : LREAL;
    AI_VoltageSHU_rezervnyi_vvod_LL : LREAL;
    AI_VoltageSHU_rezervnyi_vvod_LW : LREAL;
    AI_VoltageSHU_rezervnyi_vvod_command : UINT;
    AI_VoltageSHU_rezervnyi_vvod_newHL : LREAL;
    AI_VoltageSHU_rezervnyi_vvod_newHW : LREAL;
    AI_VoltageSHU_rezervnyi_vvod_newLL : LREAL;
    AI_VoltageSHU_rezervnyi_vvod_newLW : LREAL;
    AI_VoltageSHU_rezervnyi_vvod_status : UDINT;
    AI_VoltageSHU_rezervnyi_vvod_value : LREAL;
    AI_dP_gaza_na_konfuzore_nagnetatelia_HL : LREAL;
    AI_dP_gaza_na_konfuzore_nagnetatelia_LL : LREAL;
    AI_dP_gaza_na_konfuzore_nagnetatelia_command : UINT;
    AI_dP_gaza_na_konfuzore_nagnetatelia_newHL : LREAL;
    AI_dP_gaza_na_konfuzore_nagnetatelia_newLL : LREAL;
    AI_dP_gaza_na_konfuzore_nagnetatelia_status : UDINT;
    AI_dP_gaza_na_konfuzore_nagnetatelia_value : LREAL;
    AI_dPmaslo_gaz_HL : LREAL;
    AI_dPmaslo_gaz_LA : LREAL;
    AI_dPmaslo_gaz_LL : LREAL;
    AI_dPmaslo_gaz_LW : LREAL;
    AI_dPmaslo_gaz_command : UINT;
    AI_dPmaslo_gaz_newHL : LREAL;
    AI_dPmaslo_gaz_newLA : LREAL;
    AI_dPmaslo_gaz_newLL : LREAL;
    AI_dPmaslo_gaz_newLW : LREAL;
    AI_dPmaslo_gaz_status : UDINT;
    AI_dPmaslo_gaz_value : LREAL;
    AI_T_perednego_opornogo_podshipnika_dvigatelia_t1_HA : LREAL;
    AI_T_perednego_opornogo_podshipnika_dvigatelia_t1_HW : LREAL;
    AI_T_perednego_opornogo_podshipnika_dvigatelia_t1_newHA : LREAL;
    AI_T_perednego_opornogo_podshipnika_dvigatelia_t1_newHW : LREAL;
    AI_T_gaz_out_nagnetatelia_HA : LREAL;
    AI_T_gaz_out_nagnetatelia_HW : LREAL;
    AI_T_gaz_out_nagnetatelia_newHA : LREAL;
    AI_T_gaz_out_nagnetatelia_newHW : LREAL;
    AI_T_vnytri_shkafa_HL : LREAL;
    AI_T_vnytri_shkafa_HW : LREAL;
    AI_T_vnytri_shkafa_LL : LREAL;
    AI_T_vnytri_shkafa_LW : LREAL;
    AI_T_vnytri_shkafa_newHL : LREAL;
    AI_T_vnytri_shkafa_newHW : LREAL;
    AI_T_vnytri_shkafa_newLL : LREAL;
    AI_T_vnytri_shkafa_newLW : LREAL;
    AI_dPmaslo_gaz_newMaxChangeDown : LREAL;
    AI_dPmaslo_gaz_newMaxChangeUP : LREAL;
  END_VAR
